C01815=1076.234,414.000,-108.664,176.398,32.358,155.824
C01816=1076.246,414.386,-108.731,176.405,32.374,155.827
C01817=1076.257,414.773,-108.798,176.414,32.390,155.831
C01818=1076.269,415.159,-108.866,176.422,32.405,155.834
C01819=1076.276,415.405,-108.908,176.427,32.415,155.836
C01820=1076.283,415.651,-108.952,176.432,32.425,155.839
C01821=1076.291,415.898,-108.995,176.438,32.436,155.841
C01822=1076.298,416.143,-109.038,176.442,32.446,155.843
C01823=1076.305,416.389,-109.080,176.447,32.456,155.846
C01824=1076.313,416.636,-109.124,176.453,32.466,155.848
C01825=1076.320,416.882,-109.167,176.458,32.477,155.850
C01826=1076.327,417.128,-109.210,176.463,32.487,155.853
C01827=1076.334,417.374,-109.253,176.469,32.497,155.855
C01828=1076.342,417.620,-109.297,176.474,32.507,155.857
C01829=1076.349,417.867,-109.340,176.480,32.518,155.859
C01830=1076.356,418.112,-109.383,176.485,32.529,155.862
C01831=1076.363,418.358,-109.426,176.489,32.539,155.864
C01832=1076.371,418.605,-109.470,176.495,32.549,155.867
C01833=1076.378,418.850,-109.513,176.500,32.560,155.869
C01834=1076.386,419.097,-109.557,176.506,32.571,155.871
C01835=1076.392,419.343,-109.600,176.511,32.581,155.874
C01836=1076.400,419.589,-109.644,176.517,32.592,155.876
C01837=1076.408,419.835,-109.688,176.522,32.602,155.879
C01838=1076.415,420.081,-109.731,176.528,32.613,155.881
C01839=1076.423,420.327,-109.775,176.533,32.624,155.883
C01840=1076.430,420.573,-109.818,176.539,32.635,155.886
C01841=1076.438,420.819,-109.861,176.544,32.645,155.888
C01842=1076.446,421.066,-109.905,176.550,32.656,155.891
C01843=1076.453,421.311,-109.949,176.555,32.667,155.893
C01844=1076.460,421.557,-109.993,176.561,32.677,155.896
C01845=1076.468,421.804,-110.037,176.566,32.688,155.898
C01846=1076.475,422.049,-110.080,176.572,32.700,155.901
C01847=1076.482,422.295,-110.125,176.577,32.710,155.903
C01848=1076.490,422.542,-110.169,176.583,32.721,155.906
C01849=1076.498,422.787,-110.213,176.589,32.733,155.908
C01850=1076.505,423.034,-110.257,176.594,32.744,155.911
C01851=1076.513,423.279,-110.301,176.600,32.755,155.913
C01852=1076.520,423.525,-110.344,176.605,32.766,155.916
C01853=1076.527,423.771,-110.389,176.611,32.777,155.918
C01854=1076.535,424.017,-110.433,176.617,32.789,155.921
C01855=1076.542,424.263,-110.478,176.622,32.800,155.924
C01856=1076.550,424.508,-110.522,176.628,32.811,155.926
C01857=1076.557,424.755,-110.566,176.634,32.823,155.929
C01858=1076.565,425.001,-110.610,176.639,32.834,155.931
C01859=1076.573,425.247,-110.655,176.645,32.845,155.934
C01860=1076.580,425.493,-110.700,176.651,32.857,155.937
C01861=1076.588,425.738,-110.744,176.656,32.868,155.939
C01862=1076.595,425.984,-110.788,176.662,32.879,155.942
C01863=1076.604,426.253,-110.836,176.668,32.892,155.945
C01864=1076.612,426.521,-110.885,176.675,32.905,155.948
C01865=1076.620,426.788,-110.934,176.681,32.917,155.951
C01866=1076.629,427.057,-110.983,176.687,32.930,155.953
C01867=1076.636,427.303,-111.027,176.693,32.942,155.956
C01868=1076.644,427.548,-111.072,176.699,32.954,155.959
C01869=1076.652,427.794,-111.117,176.705,32.965,155.962
C01870=1076.660,428.040,-111.161,176.711,32.977,155.964
C01871=1076.667,428.286,-111.206,176.717,32.989,155.967
C01872=1076.674,428.532,-111.251,176.723,33.001,155.970
C01873=1076.682,428.778,-111.297,176.729,33.013,155.973
C01874=1076.690,429.023,-111.341,176.735,33.024,155.975
C01875=1076.697,429.270,-111.386,176.740,33.037,155.978
C01876=1076.705,429.515,-111.432,176.746,33.048,155.981
C01877=1076.713,429.761,-111.476,176.753,33.061,155.984
C01878=1076.721,430.006,-111.522,176.759,33.073,155.987
C01879=1076.728,430.252,-111.566,176.765,33.085,155.989
C01880=1076.736,430.498,-111.612,176.771,33.097,155.992
C01881=1076.744,430.744,-111.657,176.777,33.109,155.995
C01882=1076.752,430.989,-111.702,176.783,33.122,155.998
C01883=1076.760,431.235,-111.748,176.790,33.134,156.001
C01884=1076.767,431.481,-111.793,176.796,33.146,156.004
C01885=1076.775,431.726,-111.838,176.802,33.159,156.007
C01886=1076.784,431.972,-111.884,176.808,33.171,156.010
C01887=1076.791,432.218,-111.929,176.814,33.184,156.013
C01888=1076.799,432.464,-111.975,176.820,33.196,156.015
C01889=1076.806,432.709,-112.020,176.826,33.209,156.018
C01890=1076.814,432.955,-112.066,176.832,33.221,156.021
C01891=1076.822,433.201,-112.112,176.839,33.234,156.024
C01892=1076.830,433.446,-112.158,176.846,33.247,156.027
C01893=1076.837,433.692,-112.203,176.852,33.259,156.030
C01894=1076.845,433.937,-112.249,176.858,33.272,156.033
C01895=1076.853,434.183,-112.295,176.865,33.285,156.036
C01896=1076.861,434.429,-112.341,176.871,33.298,156.040
C01897=1076.869,434.673,-112.387,176.877,33.311,156.043
C01898=1076.877,434.920,-112.433,176.883,33.323,156.046
C01899=1076.885,435.165,-112.479,176.890,33.337,156.049
C01900=1076.892,435.410,-112.524,176.896,33.349,156.052
C01901=1076.901,435.656,-112.571,176.902,33.363,156.055
C01902=1076.909,435.901,-112.617,176.910,33.376,156.058
C01903=1076.917,436.147,-112.663,176.916,33.389,156.061
C01904=1076.925,436.392,-112.709,176.922,33.402,156.064
C01905=1076.932,436.639,-112.756,176.929,33.415,156.067
C01906=1076.940,436.884,-112.802,176.935,33.429,156.071
C01907=1076.948,437.130,-112.848,176.943,33.442,156.074
C01908=1076.956,437.374,-112.894,176.949,33.455,156.077
C01909=1076.965,437.620,-112.941,176.955,33.468,156.080
C01910=1076.973,437.865,-112.987,176.962,33.482,156.083
C01911=1076.981,438.111,-113.033,176.969,33.495,156.086
C01912=1076.989,438.356,-113.080,176.976,33.509,156.090
C01913=1076.998,438.601,-113.127,176.982,33.523,156.093
C01914=1077.005,438.848,-113.173,176.988,33.536,156.096
C01915=1077.013,439.093,-113.220,176.996,33.550,156.099
C01916=1077.022,439.338,-113.266,177.002,33.563,156.103
C01917=1077.030,439.584,-113.313,177.009,33.577,156.106
C01918=1077.037,439.829,-113.360,177.016,33.591,156.109
C01919=1077.048,440.127,-113.418,177.024,33.608,156.113
C01920=1077.057,440.426,-113.474,177.033,33.625,156.118
C01921=1077.067,440.725,-113.531,177.041,33.642,156.122
C01922=1077.078,441.024,-113.589,177.050,33.659,156.126
C01923=1077.086,441.269,-113.635,177.056,33.673,156.129
C01924=1077.093,441.515,-113.683,177.064,33.688,156.133
C01925=1077.102,441.760,-113.730,177.070,33.702,156.136
C01926=1077.110,442.006,-113.777,177.078,33.716,156.140
C01927=1077.119,442.250,-113.825,177.085,33.730,156.143
C01928=1077.127,442.496,-113.872,177.092,33.745,156.147
C01929=1077.135,442.740,-113.919,177.099,33.759,156.150
C01930=1077.143,442.986,-113.967,177.106,33.773,156.154
C01931=1077.152,443.231,-114.014,177.113,33.788,156.157
C01932=1077.159,443.477,-114.061,177.121,33.803,156.161
C01933=1077.168,443.722,-114.109,177.127,33.817,156.164
C01934=1077.176,443.967,-114.157,177.135,33.832,156.168
C01935=1077.185,444.213,-114.204,177.143,33.847,156.171
C01936=1077.193,444.458,-114.252,177.149,33.861,156.175
C01937=1077.201,444.703,-114.300,177.157,33.876,156.179
C01938=1077.210,444.948,-114.347,177.164,33.891,156.182
C01939=1077.218,445.193,-114.395,177.171,33.906,156.186
C01940=1077.226,445.438,-114.443,177.179,33.921,156.190
C01941=1077.235,445.683,-114.491,177.186,33.936,156.193
C01942=1077.243,445.928,-114.539,177.194,33.951,156.197
C01943=1077.251,446.174,-114.587,177.202,33.966,156.201
C01944=1077.259,446.419,-114.635,177.209,33.981,156.204
C01945=1077.269,446.664,-114.683,177.216,33.996,156.208
C01946=1077.277,446.909,-114.731,177.223,34.012,156.212
C01947=1077.285,447.154,-114.779,177.230,34.027,156.216
C01948=1077.293,447.399,-114.827,177.237,34.042,156.219
C01949=1077.303,447.644,-114.876,177.242,34.057,156.223
C01950=1077.311,447.890,-114.924,177.248,34.072,156.227
C01951=1077.320,448.134,-114.973,177.254,34.087,156.231
C01952=1077.329,448.379,-115.020,177.260,34.103,156.235
C01953=1077.337,448.624,-115.069,177.265,34.117,156.238
C01954=1077.345,448.869,-115.117,177.270,34.133,156.242
C01955=1077.355,449.113,-115.164,177.275,34.147,156.246
C01956=1077.367,449.358,-115.211,177.280,34.161,156.249
C01957=1077.380,449.603,-115.257,177.284,34.174,156.253
C01958=1077.394,449.849,-115.303,177.288,34.187,156.256
C01959=1077.034,449.844,-115.535,177.267,34.346,156.298
C01960=1077.019,449.599,-115.489,177.263,34.333,156.295
C01961=1077.006,449.354,-115.444,177.258,34.320,156.291
C01962=1076.995,449.108,-115.397,177.253,34.306,156.288
C01963=1076.985,448.864,-115.349,177.248,34.292,156.284
C01964=1076.976,448.619,-115.302,177.243,34.277,156.280
C01965=1076.967,448.374,-115.252,177.237,34.261,156.277
C01966=1076.959,448.130,-115.204,177.232,34.246,156.273
C01967=1076.949,447.885,-115.156,177.226,34.231,156.269
C01968=1076.941,447.640,-115.107,177.220,34.216,156.265
C01969=1076.933,447.395,-115.059,177.213,34.201,156.261
C01970=1076.924,447.150,-115.010,177.206,34.185,156.258
C01971=1076.916,446.904,-114.962,177.199,34.170,156.254
C01972=1076.907,446.660,-114.915,177.192,34.156,156.250
C01973=1076.899,446.415,-114.866,177.185,34.140,156.246
C01974=1076.891,446.170,-114.818,177.177,34.125,156.243
C01975=1076.881,445.924,-114.770,177.170,34.110,156.239
C01976=1076.873,445.679,-114.722,177.162,34.095,156.235
C01977=1076.865,445.434,-114.674,177.155,34.080,156.231
C01978=1076.857,445.189,-114.625,177.147,34.065,156.228
C01979=1076.848,444.944,-114.578,177.139,34.050,156.224
C01980=1076.840,444.699,-114.530,177.132,34.035,156.220
C01981=1076.832,444.453,-114.483,177.125,34.020,156.217
C01982=1076.823,444.208,-114.435,177.117,34.005,156.213
C01983=1076.815,443.963,-114.387,177.110,33.991,156.210
C01984=1076.806,443.718,-114.340,177.102,33.976,156.206
C01985=1076.798,443.473,-114.292,177.096,33.962,156.202
C01986=1076.789,443.228,-114.245,177.088,33.947,156.199
C01987=1076.781,442.982,-114.197,177.081,33.932,156.195
C01988=1076.773,442.737,-114.149,177.073,33.918,156.192
C01989=1076.765,442.492,-114.102,177.067,33.904,156.188
C01990=1076.756,442.246,-114.054,177.059,33.889,156.185
C01991=1076.748,442.001,-114.007,177.052,33.875,156.181
C01992=1076.740,441.756,-113.959,177.045,33.861,156.178
C01993=1076.732,441.511,-113.913,177.038,33.847,156.174
C01994=1076.723,441.265,-113.866,177.030,33.833,156.171
C01995=1076.715,441.020,-113.818,177.024,33.818,156.168
C01996=1076.706,440.739,-113.764,177.015,33.802,156.164
C01997=1076.696,440.456,-113.711,177.007,33.786,156.160
C01998=1076.687,440.175,-113.656,177.000,33.770,156.156
C01999=1076.678,439.894,-113.603,176.991,33.754,156.152
C02000=1076.669,439.649,-113.556,176.984,33.740,156.149
C02001=1076.661,439.403,-113.509,176.978,33.727,156.145
C02002=1076.653,439.158,-113.462,176.970,33.713,156.142
C02003=1076.645,438.912,-113.416,176.964,33.699,156.139
C02004=1076.636,438.667,-113.369,176.957,33.686,156.136
C02005=1076.628,438.421,-113.322,176.950,33.672,156.132
C02006=1076.620,438.176,-113.275,176.943,33.658,156.129
C02007=1076.612,437.930,-113.229,176.937,33.645,156.126
C02008=1076.604,437.685,-113.183,176.930,33.631,156.123
C02009=1076.596,437.440,-113.136,176.923,33.618,156.119
C02010=1076.587,437.194,-113.089,176.916,33.605,156.116
C02011=1076.580,436.949,-113.044,176.910,33.591,156.113
C02012=1076.571,436.703,-112.997,176.903,33.578,156.110
C02013=1076.564,436.458,-112.951,176.896,33.565,156.107
C02014=1076.556,436.212,-112.904,176.889,33.552,156.103
C02015=1076.548,435.967,-112.858,176.883,33.538,156.100
C02016=1076.539,435.721,-112.812,176.877,33.526,156.097
C02017=1076.532,435.476,-112.766,176.870,33.513,156.094
C02018=1076.523,435.230,-112.719,176.864,33.499,156.091
C02019=1076.516,434.985,-112.674,176.857,33.487,156.088
C02020=1076.508,434.739,-112.628,176.850,33.473,156.085
C02021=1076.499,434.494,-112.581,176.844,33.461,156.082
C02022=1076.492,434.248,-112.536,176.837,33.448,156.079
C02023=1076.484,434.003,-112.490,176.831,33.435,156.076
C02024=1076.476,433.757,-112.444,176.824,33.422,156.073
C02025=1076.468,433.511,-112.398,176.818,33.410,156.070
C02026=1076.461,433.266,-112.353,176.812,33.397,156.067
C02027=1076.452,433.020,-112.307,176.805,33.384,156.064
C02028=1076.445,432.774,-112.261,176.799,33.371,156.061
C02029=1076.437,432.529,-112.215,176.793,33.359,156.058
C02030=1076.429,432.283,-112.170,176.786,33.346,156.055
C02031=1076.421,432.037,-112.124,176.780,33.334,156.052
C02032=1076.414,431.792,-112.078,176.774,33.321,156.049
C02033=1076.406,431.546,-112.032,176.768,33.309,156.046
C02034=1076.398,431.301,-111.988,176.761,33.297,156.043
C02035=1076.390,431.055,-111.942,176.755,33.285,156.040
C02036=1076.382,430.809,-111.896,176.749,33.272,156.037
C02037=1076.375,430.563,-111.851,176.742,33.260,156.034
C02038=1076.366,430.318,-111.806,176.736,33.248,156.032
C02039=1076.359,430.073,-111.761,176.731,33.236,156.029
C02040=1076.351,429.826,-111.716,176.725,33.223,156.026
C02041=1076.344,429.581,-111.670,176.719,33.211,156.023
C02042=1076.336,429.335,-111.626,176.712,33.199,156.020
C02043=1076.328,429.090,-111.580,176.706,33.187,156.017
C02044=1076.320,428.843,-111.535,176.700,33.176,156.015
C02045=1076.312,428.597,-111.491,176.694,33.163,156.012
C02046=1076.304,428.352,-111.445,176.688,33.151,156.009
C02047=1076.297,428.106,-111.400,176.682,33.140,156.006
C02048=1076.290,427.860,-111.355,176.676,33.128,156.004
C02049=1076.282,427.614,-111.311,176.670,33.116,156.001
C02050=1076.274,427.368,-111.266,176.664,33.104,155.998
C02051=1076.266,427.122,-111.221,176.659,33.092,155.995
C02052=1076.258,426.853,-111.172,176.651,33.080,155.993
C02053=1076.249,426.583,-111.123,176.645,33.067,155.990
C02054=1076.240,426.314,-111.074,176.639,33.054,155.987
C02055=1076.232,426.044,-111.025,176.632,33.042,155.984
C02056=1076.225,425.798,-110.980,176.627,33.031,155.981
C02057=1076.217,425.552,-110.936,176.621,33.019,155.978
C02058=1076.210,425.307,-110.891,176.615,33.007,155.976
C02059=1076.202,425.061,-110.847,176.609,32.996,155.973
C02060=1076.194,424.814,-110.803,176.603,32.985,155.970
C02061=1076.187,424.568,-110.759,176.597,32.973,155.968
C02062=1076.179,424.323,-110.714,176.592,32.962,155.965
C02063=1076.171,424.077,-110.669,176.586,32.951,155.963
C02064=1076.164,423.831,-110.626,176.580,32.939,155.960
C02065=1076.157,423.585,-110.581,176.575,32.929,155.958
C02066=1076.149,423.339,-110.537,176.569,32.917,155.955
C02067=1076.141,423.093,-110.493,176.564,32.906,155.952
C02068=1076.134,422.847,-110.449,176.558,32.895,155.950
C02069=1076.127,422.601,-110.405,176.552,32.884,155.947
C02070=1076.119,422.355,-110.361,176.547,32.873,155.945
C02071=1076.112,422.109,-110.317,176.540,32.862,155.942
C02072=1076.104,421.863,-110.273,176.535,32.851,155.940
C02073=1076.096,421.617,-110.229,176.529,32.840,155.937
C02074=1076.090,421.371,-110.185,176.524,32.829,155.935
C02075=1076.082,421.125,-110.141,176.518,32.818,155.932
C02076=1076.074,420.879,-110.097,176.513,32.807,155.930
C02077=1076.067,420.634,-110.054,176.507,32.797,155.927
C02078=1076.059,420.387,-110.010,176.502,32.786,155.925
C02079=1076.051,420.141,-109.967,176.496,32.775,155.923
C02080=1076.044,419.895,-109.923,176.491,32.764,155.920
C02081=1076.037,419.648,-109.879,176.485,32.754,155.918
C02082=1076.030,419.403,-109.836,176.480,32.743,155.915
C02083=1076.022,419.156,-109.792,176.474,32.733,155.913
C02084=1076.014,418.910,-109.749,176.469,32.722,155.911
C02085=1076.007,418.664,-109.705,176.463,32.711,155.908
C02086=1076.000,418.418,-109.662,176.458,32.701,155.906
C02087=1075.992,418.172,-109.618,176.453,32.691,155.903
C02088=1075.985,417.926,-109.575,176.447,32.680,155.901
C02089=1075.977,417.680,-109.532,176.442,32.670,155.899
C02090=1075.970,417.434,-109.488,176.436,32.660,155.896
C02091=1075.963,417.188,-109.445,176.431,32.649,155.894
C02092=1075.956,416.942,-109.402,176.426,32.639,155.892
C02093=1075.948,416.696,-109.359,176.421,32.628,155.889
C02094=1075.941,416.450,-109.315,176.416,32.618,155.887
C02095=1075.933,416.203,-109.272,176.411,32.608,155.885
C02096=1075.926,415.957,-109.229,176.405,32.598,155.882
C02097=1075.919,415.712,-109.186,176.400,32.587,155.880
C02098=1075.911,415.465,-109.143,176.395,32.578,155.878
C02099=1075.904,415.219,-109.100,176.389,32.567,155.876
C02100=1075.897,414.973,-109.057,176.384,32.557,155.873
C02101=1075.890,414.726,-109.014,176.379,32.547,155.871
C02102=1075.882,414.480,-108.972,176.374,32.537,155.869
C02103=1075.875,414.234,-108.929,176.368,32.527,155.867
C02104=1075.867,413.988,-108.885,176.363,32.517,155.864
C02105=1075.861,413.741,-108.843,176.358,32.507,155.862
C02106=1075.853,413.495,-108.801,176.354,32.497,155.860
C02107=1075.845,413.249,-108.757,176.348,32.487,155.858
C02108=1075.838,412.997,-108.714,176.343,32.478,155.856
C02109=1075.831,412.745,-108.671,176.338,32.468,155.853
C02110=1075.823,412.493,-108.627,176.332,32.458,155.851
C02111=1075.816,412.241,-108.583,176.327,32.448,155.849
C02112=1075.809,411.995,-108.541,176.322,32.438,155.847
C02113=1075.801,411.749,-108.499,176.317,32.429,155.845
C02114=1075.794,411.502,-108.456,176.312,32.419,155.842
C02115=1075.787,411.255,-108.413,176.307,32.409,155.840
C02116=1075.779,411.010,-108.371,176.302,32.399,155.838
C02117=1075.773,410.763,-108.329,176.297,32.390,155.836
C02118=1075.766,410.517,-108.286,176.292,32.380,155.834
C02119=1075.758,410.271,-108.244,176.287,32.371,155.832
C02120=1075.751,410.025,-108.202,176.282,32.361,155.830
C02121=1075.744,409.778,-108.159,176.277,32.352,155.828
C02122=1075.736,409.532,-108.117,176.272,32.342,155.826
C02123=1075.730,409.285,-108.075,176.267,32.333,155.823
C02124=1075.722,409.039,-108.033,176.262,32.323,155.821
C02125=1075.715,408.793,-107.991,176.257,32.314,155.819
C02126=1075.708,408.546,-107.948,176.252,32.305,155.817
C02127=1075.701,408.300,-107.907,176.247,32.295,155.815
C02128=1075.694,408.053,-107.864,176.243,32.286,155.813
C02129=1075.687,407.807,-107.822,176.238,32.276,155.811
C02130=1075.680,407.561,-107.781,176.233,32.268,155.809
C02131=1075.673,407.314,-107.738,176.228,32.258,155.807
C02132=1075.667,407.068,-107.697,176.223,32.249,155.805
C02133=1075.660,406.822,-107.655,176.219,32.240,155.803
C02134=1075.652,406.575,-107.613,176.214,32.230,155.801
C02135=1075.645,406.329,-107.571,176.209,32.221,155.799
C02136=1075.638,406.083,-107.530,176.204,32.213,155.797
C02137=1075.631,405.837,-107.488,176.199,32.203,155.795
C02138=1075.624,405.590,-107.446,176.195,32.194,155.793
C02139=1075.617,405.343,-107.405,176.190,32.185,155.791
C02140=1075.609,405.097,-107.363,176.185,32.176,155.789
C02141=1075.603,404.850,-107.321,176.180,32.167,155.787
C02142=1075.595,404.604,-107.280,176.175,32.158,155.785
C02143=1075.589,404.358,-107.239,176.171,32.149,155.783
C02144=1075.582,404.111,-107.196,176.166,32.141,155.781
C02145=1075.575,403.865,-107.155,176.162,32.132,155.779
C02146=1075.567,403.618,-107.114,176.157,32.123,155.777
C02147=1075.560,403.372,-107.073,176.152,32.114,155.775
C02148=1075.554,403.125,-107.031,176.148,32.105,155.774
C02149=1075.547,402.879,-106.990,176.143,32.096,155.772
C02150=1075.539,402.632,-106.949,176.138,32.088,155.770
C02151=1075.532,402.386,-106.907,176.133,32.079,155.768
C02152=1075.525,402.139,-106.866,176.129,32.070,155.766
C02153=1075.518,401.893,-106.825,176.124,32.062,155.764
C02154=1075.512,401.646,-106.784,176.120,32.053,155.762
C02155=1075.504,401.400,-106.742,176.115,32.044,155.760
C02156=1075.498,401.154,-106.701,176.111,32.035,155.759
C02157=1075.490,400.907,-106.660,176.106,32.027,155.757
C02158=1075.483,400.661,-106.619,176.101,32.019,155.755
C02159=1075.477,400.414,-106.579,176.096,32.010,155.753
C02160=1075.470,400.179,-106.539,176.093,32.002,155.751
C02161=1075.464,399.943,-106.500,176.088,31.994,155.750
C02162=1075.456,399.708,-106.461,176.084,31.986,155.748
C02163=1075.450,399.472,-106.422,176.079,31.978,155.746
C02164=1075.443,399.237,-106.382,176.075,31.970,155.744
C02165=1075.437,399.001,-106.343,176.071,31.961,155.743
C02166=1075.430,398.765,-106.305,176.066,31.953,155.741
C02167=1075.421,398.432,-106.250,176.060,31.942,155.738
C02168=1075.414,398.186,-106.209,176.056,31.934,155.737
C02169=1075.407,397.939,-106.168,176.051,31.925,155.735
C02170=1075.400,397.692,-106.127,176.047,31.917,155.733
C02171=1075.393,397.446,-106.087,176.043,31.909,155.731
C02172=1075.386,397.199,-106.046,176.038,31.901,155.730
C02173=1075.380,396.953,-106.006,176.033,31.892,155.728
C02174=1075.372,396.706,-105.964,176.029,31.885,155.726
C02175=1075.366,396.460,-105.924,176.025,31.876,155.724
C02176=1075.358,396.213,-105.884,176.020,31.868,155.723
C02177=1075.351,395.967,-105.843,176.015,31.860,155.721
C02178=1075.345,395.720,-105.803,176.012,31.852,155.719
C02179=1075.338,395.473,-105.763,176.007,31.844,155.717
C02180=1075.331,395.227,-105.722,176.002,31.835,155.716
C02181=1075.324,394.980,-105.681,175.998,31.827,155.714
C02182=1075.317,394.734,-105.642,175.994,31.819,155.712
C02183=1075.311,394.487,-105.602,175.989,31.811,155.711
C02184=1075.304,394.240,-105.561,175.985,31.803,155.709
C02185=1075.297,393.994,-105.520,175.981,31.795,155.707
C02186=1075.290,393.747,-105.480,175.976,31.787,155.705
C02187=1075.283,393.501,-105.440,175.972,31.779,155.704
C02188=1075.277,393.254,-105.400,175.968,31.772,155.702
C02189=1075.269,393.007,-105.360,175.963,31.764,155.701
C02190=1075.263,392.761,-105.320,175.959,31.756,155.699
C02191=1075.256,392.514,-105.280,175.954,31.748,155.697
C02192=1075.249,392.268,-105.240,175.950,31.740,155.695
C02193=1075.242,392.021,-105.200,175.946,31.732,155.694
C02194=1075.236,391.774,-105.160,175.941,31.724,155.692
C02195=1075.229,391.528,-105.120,175.937,31.716,155.691
C02196=1075.222,391.282,-105.080,175.933,31.709,155.689
C02197=1075.215,391.034,-105.041,175.928,31.701,155.687
C02198=1075.208,390.788,-105.001,175.924,31.694,155.686
C02199=1075.201,390.541,-104.961,175.920,31.686,155.684
C02200=1075.195,390.295,-104.921,175.915,31.678,155.683
C02201=1075.187,390.048,-104.881,175.912,31.670,155.681
C02202=1075.181,389.801,-104.842,175.907,31.663,155.679
C02203=1075.174,389.555,-104.802,175.902,31.655,155.678
C02204=1075.167,389.308,-104.763,175.899,31.648,155.676
C02205=1075.161,389.061,-104.723,175.894,31.640,155.675
C02206=1075.153,388.814,-104.683,175.890,31.633,155.673
C02207=1075.147,388.568,-104.643,175.886,31.625,155.671
C02208=1075.140,388.321,-104.604,175.881,31.617,155.670
C02209=1075.133,388.075,-104.565,175.877,31.610,155.668
C02210=1075.127,387.828,-104.525,175.873,31.603,155.667
C02211=1075.120,387.582,-104.486,175.869,31.595,155.665
C02212=1075.113,387.335,-104.447,175.864,31.588,155.664
C02213=1075.106,387.088,-104.407,175.861,31.580,155.662
C02214=1075.100,386.841,-104.368,175.856,31.573,155.661
C02215=1075.093,386.595,-104.328,175.852,31.565,155.659
C02216=1075.086,386.354,-104.290,175.848,31.558,155.658
C02217=1075.080,386.114,-104.252,175.844,31.551,155.656
C02218=1075.074,385.874,-104.214,175.839,31.544,155.655
C02219=1075.067,385.633,-104.175,175.836,31.537,155.653
C02220=1075.060,385.394,-104.137,175.832,31.530,155.652
C02221=1075.054,385.153,-104.099,175.828,31.522,155.650
C02222=1075.047,384.913,-104.060,175.824,31.515,155.649
C02223=1075.041,384.672,-104.022,175.819,31.508,155.647
C02224=1075.034,384.425,-103.983,175.816,31.501,155.646
C02225=1075.027,384.179,-103.944,175.811,31.494,155.644
C02226=1075.021,383.932,-103.905,175.807,31.486,155.643
C02227=1075.015,383.686,-103.866,175.804,31.479,155.641
C02228=1075.008,383.439,-103.827,175.799,31.472,155.640
C02229=1075.001,383.192,-103.788,175.795,31.464,155.638
C02230=1074.995,382.945,-103.749,175.791,31.457,155.637
C02231=1074.988,382.698,-103.710,175.787,31.451,155.635
C02232=1074.981,382.451,-103.671,175.782,31.443,155.634
C02233=1074.974,382.204,-103.632,175.779,31.436,155.632
C02234=1074.968,381.957,-103.593,175.774,31.429,155.631
C02235=1074.962,381.711,-103.555,175.771,31.422,155.629
C02236=1074.955,381.464,-103.516,175.766,31.415,155.628
C02237=1074.949,381.218,-103.477,175.762,31.408,155.627
C02238=1074.942,380.971,-103.438,175.759,31.401,155.625
C02239=1074.935,380.724,-103.399,175.754,31.394,155.624
C02240=1074.928,380.477,-103.360,175.750,31.387,155.622
C02241=1074.922,380.230,-103.322,175.746,31.380,155.621
C02242=1074.915,379.983,-103.283,175.742,31.373,155.619
C02243=1074.909,379.737,-103.245,175.739,31.366,155.618
C02244=1074.902,379.490,-103.206,175.734,31.359,155.617
C02245=1074.895,379.243,-103.169,175.730,31.352,155.615
C02246=1074.888,378.996,-103.130,175.726,31.345,155.614
C02247=1074.881,378.749,-103.091,175.722,31.338,155.612
C02248=1074.875,378.502,-103.053,175.719,31.332,155.611
C02249=1074.868,378.256,-103.014,175.714,31.324,155.610
C02250=1074.862,378.008,-102.976,175.710,31.318,155.608
C02251=1074.855,377.761,-102.937,175.706,31.311,155.607
C02252=1074.849,377.515,-102.899,175.702,31.304,155.605
C02253=1074.842,377.268,-102.861,175.698,31.298,155.604
C02254=1074.835,377.021,-102.822,175.694,31.291,155.603
C02255=1074.829,376.773,-102.784,175.690,31.284,155.601
C02256=1074.823,376.527,-102.745,175.687,31.277,155.600
C02257=1074.815,376.280,-102.708,175.682,31.270,155.599
C02258=1074.809,376.033,-102.670,175.678,31.264,155.597
C02259=1074.803,375.787,-102.631,175.675,31.257,155.596
C02260=1074.796,375.539,-102.593,175.670,31.250,155.595
C02261=1074.789,375.292,-102.554,175.667,31.243,155.593
C02262=1074.783,375.046,-102.516,175.663,31.237,155.592
C02263=1074.777,374.798,-102.478,175.658,31.230,155.590
C02264=1074.771,374.551,-102.441,175.655,31.223,155.589
C02265=1074.764,374.305,-102.402,175.651,31.217,155.588
C02266=1074.757,374.057,-102.364,175.648,31.210,155.586
C02267=1074.751,373.811,-102.326,175.643,31.203,155.585
C02268=1074.745,373.563,-102.288,175.639,31.197,155.584
C02269=1074.738,373.317,-102.250,175.636,31.191,155.583
C02270=1074.731,373.070,-102.212,175.631,31.183,155.581
C02271=1074.725,372.823,-102.174,175.628,31.177,155.580
C02272=1074.718,372.597,-102.140,175.624,31.171,155.579
C02273=1074.713,372.371,-102.105,175.620,31.165,155.578
C02274=1074.707,372.145,-102.072,175.617,31.159,155.576
C02275=1074.701,371.920,-102.037,175.613,31.153,155.575
C02276=1074.695,371.694,-102.002,175.610,31.148,155.574
C02277=1074.689,371.468,-101.968,175.607,31.142,155.573
C02278=1074.683,371.243,-101.933,175.603,31.136,155.572
C02279=1074.677,371.017,-101.898,175.600,31.130,155.570
C02280=1074.670,370.770,-101.861,175.596,31.124,155.569
C02281=1074.664,370.523,-101.823,175.591,31.117,155.568
C02282=1074.657,370.276,-101.787,175.588,31.111,155.567
C02283=1074.651,370.028,-101.748,175.584,31.104,155.565
C02284=1074.644,369.782,-101.711,175.581,31.098,155.564
C02285=1074.638,369.535,-101.673,175.576,31.092,155.563
C02286=1074.631,369.288,-101.636,175.572,31.086,155.562
C02287=1074.625,369.041,-101.598,175.569,31.079,155.560
C02288=1074.618,368.794,-101.561,175.565,31.073,155.559
C02289=1074.612,368.546,-101.523,175.562,31.067,155.558
C02290=1074.605,368.300,-101.486,175.557,31.060,155.557
C02291=1074.600,368.052,-101.449,175.554,31.054,155.555
C02292=1074.592,367.805,-101.412,175.550,31.048,155.554
C02293=1074.586,367.559,-101.374,175.546,31.041,155.553
C02294=1074.579,367.311,-101.337,175.543,31.035,155.552
C02295=1074.574,367.064,-101.299,175.538,31.029,155.550
C02296=1074.567,366.818,-101.262,175.535,31.023,155.549
C02297=1074.561,366.570,-101.225,175.531,31.016,155.548
C02298=1074.554,366.323,-101.188,175.527,31.010,155.547
C02299=1074.548,366.076,-101.151,175.524,31.004,155.546
C02300=1074.541,365.829,-101.113,175.519,30.998,155.544
C02301=1074.536,365.581,-101.076,175.516,30.992,155.543
C02302=1074.529,365.335,-101.039,175.512,30.985,155.542
C02303=1074.522,365.087,-101.002,175.509,30.979,155.541
C02304=1074.516,364.840,-100.964,175.505,30.973,155.540
C02305=1074.510,364.593,-100.928,175.501,30.967,155.538
C02306=1074.503,364.345,-100.891,175.498,30.961,155.537
C02307=1074.497,364.099,-100.853,175.493,30.955,155.536
C02308=1074.491,363.852,-100.817,175.490,30.949,155.535
C02309=1074.484,363.604,-100.780,175.486,30.943,155.534
C02310=1074.477,363.357,-100.743,175.483,30.937,155.532
C02311=1074.471,363.110,-100.706,175.479,30.931,155.531
C02312=1074.465,362.862,-100.669,175.475,30.925,155.530
C02313=1074.458,362.615,-100.632,175.472,30.919,155.529
C02314=1074.452,362.368,-100.596,175.467,30.913,155.528
C02315=1074.445,362.122,-100.559,175.464,30.907,155.527
C02316=1074.438,361.874,-100.522,175.460,30.901,155.525
C02317=1074.433,361.627,-100.485,175.457,30.895,155.524
C02318=1074.426,361.380,-100.449,175.453,30.889,155.523
C02319=1074.420,361.133,-100.412,175.449,30.883,155.522
C02320=1074.413,360.885,-100.375,175.446,30.877,155.521
C02321=1074.407,360.638,-100.339,175.442,30.871,155.520
C02322=1074.400,360.391,-100.302,175.439,30.865,155.518
C02323=1074.394,360.144,-100.266,175.434,30.859,155.517
C02324=1074.388,359.896,-100.229,175.431,30.853,155.516
C02325=1074.382,359.649,-100.193,175.427,30.848,155.515
C02326=1074.375,359.401,-100.156,175.424,30.842,155.514
C02327=1074.369,359.154,-100.119,175.420,30.836,155.513
C02328=1074.363,358.937,-100.088,175.417,30.831,155.512
C02329=1074.357,358.720,-100.055,175.414,30.826,155.511
C02330=1074.352,358.503,-100.024,175.410,30.821,155.510
C02331=1074.346,358.285,-99.991,175.407,30.815,155.509
C02332=1074.340,358.068,-99.960,175.404,30.810,155.508
C02333=1074.335,357.850,-99.928,175.401,30.805,155.507
C02334=1074.329,357.633,-99.895,175.398,30.800,155.506
C02335=1074.324,357.416,-99.863,175.395,30.795,155.505
C02336=1074.317,357.168,-99.827,175.391,30.790,155.504
C02337=1074.311,356.921,-99.791,175.387,30.783,155.503
C02338=1074.305,356.674,-99.754,175.383,30.778,155.502
C02339=1074.298,356.426,-99.718,175.380,30.772,155.501
C02340=1074.292,356.179,-99.682,175.376,30.766,155.499
C02341=1074.285,355.932,-99.646,175.373,30.760,155.498
C02342=1074.279,355.685,-99.610,175.369,30.755,155.497
C02343=1074.273,355.437,-99.574,175.366,30.750,155.496
C02344=1074.267,355.190,-99.538,175.362,30.744,155.495
C02345=1074.260,354.943,-99.501,175.358,30.738,155.494
C02346=1074.254,354.696,-99.466,175.355,30.732,155.493
C02347=1074.248,354.448,-99.429,175.351,30.727,155.492
C02348=1074.242,354.201,-99.393,175.348,30.721,155.491
C02349=1074.236,353.954,-99.357,175.344,30.715,155.490
C02350=1074.229,353.706,-99.322,175.341,30.710,155.489
C02351=1074.222,353.459,-99.285,175.337,30.704,155.488
C02352=1074.216,353.212,-99.250,175.334,30.698,155.486
C02353=1074.210,352.965,-99.213,175.330,30.693,155.485
C02354=1074.204,352.717,-99.177,175.326,30.687,155.484
C02355=1074.198,352.469,-99.142,175.323,30.682,155.483
C02356=1074.191,352.223,-99.106,175.319,30.676,155.482
C02357=1074.185,351.975,-99.070,175.316,30.670,155.481
C02358=1074.179,351.727,-99.034,175.312,30.665,155.480
C02359=1074.172,351.480,-98.999,175.309,30.659,155.479
C02360=1074.166,351.233,-98.963,175.305,30.654,155.478
C02361=1074.160,350.985,-98.927,175.302,30.648,155.477
C02362=1074.153,350.738,-98.892,175.298,30.643,155.476
C02363=1074.147,350.491,-98.856,175.295,30.638,155.475
C02364=1074.141,350.243,-98.820,175.292,30.632,155.474
C02365=1074.134,349.996,-98.785,175.288,30.627,155.473
C02366=1074.128,349.749,-98.749,175.285,30.621,155.472
C02367=1074.122,349.501,-98.714,175.281,30.616,155.471
C02368=1074.116,349.254,-98.678,175.278,30.610,155.470
C02369=1074.109,349.007,-98.642,175.274,30.605,155.469
C02370=1074.102,348.759,-98.607,175.271,30.600,155.468
C02371=1074.096,348.511,-98.571,175.267,30.594,155.467
C02372=1074.091,348.265,-98.536,175.264,30.589,155.466
C02373=1074.084,348.017,-98.501,175.260,30.583,155.465
C02374=1074.078,347.769,-98.465,175.256,30.578,155.464
C02375=1074.071,347.522,-98.430,175.253,30.572,155.463
C02376=1074.065,347.274,-98.394,175.249,30.567,155.462
C02377=1074.059,347.027,-98.359,175.247,30.562,155.461
C02378=1074.053,346.780,-98.324,175.243,30.556,155.460
C02379=1074.046,346.533,-98.288,175.240,30.551,155.459
C02380=1074.041,346.284,-98.253,175.236,30.545,155.458
C02381=1074.035,346.037,-98.218,175.233,30.540,155.457
C02382=1074.029,345.790,-98.183,175.229,30.535,155.456
C02383=1074.022,345.543,-98.148,175.226,30.529,155.455
C02384=1074.017,345.327,-98.117,175.223,30.525,155.454
C02385=1074.011,345.112,-98.086,175.219,30.520,155.453
C02386=1074.005,344.896,-98.056,175.217,30.516,155.452
C02387=1074.001,344.680,-98.025,175.214,30.511,155.451
C02388=1073.995,344.464,-97.994,175.211,30.506,155.450
C02389=1073.989,344.249,-97.963,175.208,30.502,155.449
C02390=1073.984,344.033,-97.933,175.205,30.497,155.449
C02391=1073.979,343.817,-97.902,175.202,30.492,155.448
C02392=1073.972,343.570,-97.867,175.198,30.487,155.447
C02393=1073.966,343.321,-97.832,175.195,30.482,155.446
C02394=1073.960,343.075,-97.797,175.192,30.477,155.445
C02395=1073.953,342.827,-97.762,175.189,30.472,155.444
C02396=1073.947,342.579,-97.728,175.185,30.467,155.443
C02397=1073.941,342.332,-97.693,175.181,30.462,155.442
C02398=1073.935,342.084,-97.658,175.178,30.456,155.441
C02399=1073.928,341.837,-97.623,175.174,30.451,155.440
C02400=1073.922,341.590,-97.589,175.171,30.446,155.439
C02401=1073.916,341.342,-97.553,175.168,30.441,155.438
C02402=1073.910,341.094,-97.519,175.165,30.436,155.437
C02403=1073.904,340.848,-97.484,175.161,30.430,155.436
C02404=1073.897,340.600,-97.450,175.158,30.425,155.435
C02405=1073.891,340.352,-97.414,175.154,30.420,155.434
C02406=1073.885,340.105,-97.380,175.152,30.415,155.433
C02407=1073.879,339.857,-97.345,175.148,30.410,155.432
C02408=1073.873,339.610,-97.311,175.145,30.405,155.432
C02409=1073.867,339.362,-97.276,175.141,30.399,155.431
C02410=1073.860,339.114,-97.240,175.137,30.394,155.430
C02411=1073.854,338.867,-97.206,175.134,30.389,155.429
C02412=1073.848,338.620,-97.171,175.131,30.384,155.428
C02413=1073.842,338.372,-97.137,175.128,30.379,155.427
C02414=1073.836,338.124,-97.102,175.124,30.374,155.426
C02415=1073.830,337.877,-97.068,175.121,30.369,155.425
C02416=1073.823,337.629,-97.033,175.118,30.364,155.424
C02417=1073.817,337.382,-96.999,175.115,30.359,155.423
C02418=1073.811,337.134,-96.965,175.111,30.354,155.422
C02419=1073.805,336.886,-96.930,175.108,30.349,155.421
C02420=1073.799,336.639,-96.896,175.104,30.344,155.420
C02421=1073.792,336.391,-96.862,175.102,30.339,155.419
C02422=1073.786,336.144,-96.827,175.098,30.334,155.418
C02423=1073.780,335.896,-96.792,175.095,30.329,155.418
C02424=1073.774,335.649,-96.758,175.091,30.324,155.417
C02425=1073.767,335.401,-96.724,175.088,30.319,155.416
C02426=1073.761,335.154,-96.690,175.085,30.314,155.415
C02427=1073.755,334.906,-96.656,175.081,30.309,155.414
C02428=1073.749,334.658,-96.621,175.078,30.304,155.413
C02429=1073.743,334.410,-96.587,175.075,30.299,155.412
C02430=1073.737,334.163,-96.553,175.072,30.294,155.411
C02431=1073.731,333.916,-96.519,175.068,30.289,155.410
C02432=1073.724,333.668,-96.485,175.065,30.284,155.409
C02433=1073.719,333.421,-96.450,175.062,30.279,155.409
C02434=1073.712,333.173,-96.416,175.059,30.274,155.408
C02435=1073.706,332.925,-96.382,175.055,30.269,155.407
C02436=1073.700,332.677,-96.348,175.052,30.264,155.406
C02437=1073.693,332.430,-96.315,175.049,30.260,155.405
C02438=1073.688,332.182,-96.281,175.046,30.255,155.404
C02439=1073.681,331.934,-96.246,175.042,30.250,155.403
C02440=1073.676,331.716,-96.217,175.039,30.245,155.402
C02441=1073.671,331.498,-96.186,175.037,30.241,155.402
C02442=1073.666,331.280,-96.156,175.034,30.237,155.401
C02443=1073.660,331.062,-96.126,175.031,30.232,155.400
C02444=1073.655,330.844,-96.096,175.028,30.228,155.399
C02445=1073.649,330.625,-96.067,175.025,30.224,155.399
C02446=1073.643,330.407,-96.037,175.022,30.219,155.398
C02447=1073.638,330.189,-96.008,175.019,30.216,155.397
C02448=1073.631,329.940,-95.974,175.016,30.211,155.396
C02449=1073.625,329.693,-95.940,175.013,30.206,155.395
C02450=1073.618,329.445,-95.906,175.010,30.201,155.395
C02451=1073.613,329.198,-95.873,175.006,30.196,155.394
C02452=1073.606,328.951,-95.839,175.004,30.192,155.393
C02453=1073.600,328.703,-95.805,175.000,30.187,155.392
C02454=1073.593,328.455,-95.772,174.997,30.182,155.391
C02455=1073.588,328.208,-95.738,174.994,30.178,155.390
C02456=1073.581,327.959,-95.705,174.990,30.172,155.389
C02457=1073.575,327.712,-95.671,174.987,30.168,155.389
C02458=1073.569,327.464,-95.637,174.984,30.163,155.388
C02459=1073.562,327.217,-95.604,174.981,30.159,155.387
C02460=1073.557,326.969,-95.570,174.977,30.154,155.386
C02461=1073.550,326.722,-95.537,174.975,30.149,155.385
C02462=1073.544,326.474,-95.503,174.971,30.144,155.384
C02463=1073.538,326.225,-95.470,174.968,30.140,155.384
C02464=1073.532,325.978,-95.436,174.965,30.135,155.383
C02465=1073.525,325.731,-95.404,174.962,30.130,155.382
C02466=1073.519,325.483,-95.369,174.958,30.126,155.381
C02467=1073.513,325.235,-95.336,174.956,30.121,155.380
C02468=1073.507,324.987,-95.303,174.952,30.116,155.379
C02469=1073.500,324.740,-95.270,174.950,30.111,155.378
C02470=1073.495,324.492,-95.236,174.946,30.107,155.378
C02471=1073.488,324.244,-95.203,174.943,30.102,155.377
C02472=1073.482,323.996,-95.170,174.940,30.098,155.376
C02473=1073.476,323.749,-95.136,174.936,30.093,155.375
C02474=1073.470,323.501,-95.103,174.933,30.088,155.374
C02475=1073.464,323.254,-95.070,174.930,30.084,155.374
C02476=1073.458,323.006,-95.037,174.927,30.079,155.373
C02477=1073.451,322.758,-95.003,174.924,30.074,155.372
C02478=1073.446,322.510,-94.970,174.921,30.070,155.371
C02479=1073.439,322.262,-94.937,174.917,30.065,155.370
C02480=1073.434,322.015,-94.904,174.915,30.060,155.369
C02481=1073.428,321.767,-94.871,174.911,30.055,155.368
C02482=1073.421,321.519,-94.838,174.909,30.051,155.368
C02483=1073.416,321.271,-94.805,174.905,30.046,155.367
C02484=1073.409,321.024,-94.772,174.902,30.041,155.366
C02485=1073.404,320.777,-94.738,174.899,30.037,155.365
C02486=1073.397,320.529,-94.705,174.896,30.032,155.364
C02487=1073.392,320.281,-94.672,174.893,30.027,155.364
C02488=1073.385,320.033,-94.639,174.890,30.023,155.363
C02489=1073.379,319.785,-94.606,174.887,30.019,155.362
C02490=1073.373,319.537,-94.573,174.884,30.013,155.361
C02491=1073.367,319.290,-94.540,174.880,30.009,155.360
C02492=1073.361,319.042,-94.507,174.877,30.005,155.360
C02493=1073.355,318.794,-94.475,174.874,30.000,155.359
C02494=1073.349,318.546,-94.442,174.871,29.995,155.358
C02495=1073.343,318.298,-94.409,174.868,29.991,155.357
C02496=1073.338,318.077,-94.380,174.865,29.986,155.356
C02497=1073.333,317.856,-94.349,174.863,29.982,155.356
C02498=1073.328,317.634,-94.321,174.860,29.978,155.355
C02499=1073.322,317.413,-94.291,174.858,29.974,155.354
C02500=1073.317,317.192,-94.262,174.854,29.970,155.354
C02501=1073.311,316.970,-94.233,174.852,29.966,155.353
C02502=1073.306,316.749,-94.203,174.849,29.962,155.352
C02503=1073.300,316.527,-94.174,174.846,29.958,155.351
C02504=1073.295,316.280,-94.141,174.843,29.953,155.350
C02505=1073.289,316.031,-94.109,174.840,29.949,155.350
C02506=1073.283,315.784,-94.076,174.837,29.944,155.349
C02507=1073.278,315.537,-94.043,174.834,29.939,155.348
C02508=1073.272,315.288,-94.011,174.831,29.935,155.347
C02509=1073.265,315.041,-93.978,174.828,29.930,155.346
C02510=1073.260,314.793,-93.945,174.825,29.926,155.346
C02511=1073.254,314.545,-93.912,174.822,29.921,155.345
C02512=1073.248,314.297,-93.880,174.819,29.916,155.344
C02513=1073.241,314.049,-93.847,174.816,29.912,155.343
C02514=1073.235,313.801,-93.815,174.813,29.908,155.343
C02515=1073.229,313.554,-93.782,174.810,29.904,155.342
C02516=1073.223,313.305,-93.750,174.807,29.899,155.341
C02517=1073.216,313.058,-93.718,174.804,29.895,155.340
C02518=1073.210,312.810,-93.686,174.801,29.890,155.339
C02519=1073.204,312.563,-93.654,174.798,29.886,155.339
C02520=1073.198,312.315,-93.622,174.795,29.881,155.338
C02521=1073.192,312.067,-93.589,174.792,29.877,155.337
C02522=1073.186,311.819,-93.557,174.788,29.873,155.336
C02523=1073.180,311.571,-93.524,174.786,29.868,155.336
C02524=1073.173,311.323,-93.493,174.782,29.864,155.335
C02525=1073.167,311.076,-93.460,174.780,29.860,155.334
C02526=1073.161,310.828,-93.428,174.776,29.855,155.333
C02527=1073.155,310.579,-93.396,174.774,29.851,155.333
C02528=1073.149,310.333,-93.364,174.770,29.847,155.332
C02529=1073.143,310.084,-93.332,174.768,29.842,155.331
C02530=1073.136,309.836,-93.300,174.764,29.838,155.330
C02531=1073.130,309.589,-93.268,174.762,29.833,155.330
C02532=1073.124,309.341,-93.236,174.758,29.829,155.329
C02533=1073.119,309.093,-93.204,174.756,29.825,155.328
C02534=1073.112,308.846,-93.171,174.752,29.820,155.327
C02535=1073.106,308.598,-93.140,174.750,29.816,155.327
C02536=1073.100,308.349,-93.108,174.746,29.811,155.326
C02537=1073.094,308.101,-93.076,174.744,29.807,155.325
C02538=1073.088,307.854,-93.043,174.740,29.803,155.324
C02539=1073.082,307.606,-93.011,174.738,29.798,155.324
C02540=1073.075,307.358,-92.980,174.735,29.794,155.323
C02541=1073.070,307.111,-92.948,174.732,29.790,155.322
C02542=1073.064,306.862,-92.916,174.729,29.786,155.321
C02543=1073.058,306.614,-92.884,174.726,29.781,155.321
C02544=1073.051,306.367,-92.852,174.723,29.777,155.320
C02545=1073.045,306.119,-92.820,174.720,29.772,155.319
C02546=1073.040,305.871,-92.788,174.717,29.768,155.318
C02547=1073.034,305.623,-92.756,174.714,29.764,155.318
C02548=1073.027,305.376,-92.725,174.711,29.759,155.317
C02549=1073.021,305.128,-92.693,174.709,29.755,155.316
C02550=1073.015,304.879,-92.661,174.705,29.751,155.315
C02551=1073.009,304.632,-92.630,174.702,29.746,155.315
C02552=1073.004,304.412,-92.601,174.700,29.743,155.314
C02553=1072.999,304.193,-92.573,174.697,29.739,155.313
C02554=1072.993,303.973,-92.545,174.695,29.735,155.313
C02555=1072.988,303.753,-92.518,174.692,29.731,155.312
C02556=1072.983,303.533,-92.489,174.689,29.727,155.311
C02557=1072.978,303.314,-92.461,174.686,29.723,155.311
C02558=1072.973,303.094,-92.433,174.684,29.719,155.310
C02559=1072.967,302.874,-92.405,174.681,29.715,155.309
C02560=1072.961,302.626,-92.373,174.678,29.711,155.309
C02561=1072.955,302.378,-92.342,174.676,29.707,155.308
C02562=1072.949,302.130,-92.310,174.672,29.703,155.307
C02563=1072.944,301.882,-92.279,174.670,29.698,155.306
C02564=1072.937,301.635,-92.247,174.666,29.694,155.306
C02565=1072.932,301.387,-92.216,174.664,29.690,155.305
C02566=1072.926,301.139,-92.184,174.661,29.685,155.304
C02567=1072.920,300.891,-92.153,174.658,29.681,155.303
C02568=1072.914,300.643,-92.121,174.655,29.677,155.303
C02569=1072.909,300.395,-92.090,174.652,29.672,155.302
C02570=1072.902,300.147,-92.058,174.649,29.668,155.301
C02571=1072.897,299.899,-92.027,174.647,29.664,155.301
C02572=1072.890,299.651,-91.996,174.643,29.659,155.300
C02573=1072.885,299.404,-91.964,174.641,29.655,155.299
C02574=1072.879,299.155,-91.933,174.638,29.651,155.298
C02575=1072.873,298.908,-91.902,174.635,29.647,155.298
C02576=1072.867,298.660,-91.870,174.632,29.642,155.297
C02577=1072.862,298.411,-91.839,174.630,29.638,155.296
C02578=1072.856,298.164,-91.808,174.626,29.634,155.295
C02579=1072.850,297.916,-91.776,174.624,29.629,155.295
C02580=1072.844,297.668,-91.745,174.621,29.625,155.294
C02581=1072.838,297.420,-91.713,174.618,29.621,155.293
C02582=1072.832,297.172,-91.683,174.615,29.616,155.292
C02583=1072.826,296.924,-91.651,174.612,29.612,155.292
C02584=1072.820,296.676,-91.621,174.609,29.608,155.291
C02585=1072.814,296.428,-91.589,174.607,29.604,155.290
C02586=1072.809,296.180,-91.558,174.603,29.599,155.290
C02587=1072.802,295.932,-91.527,174.601,29.596,155.289
C02588=1072.796,295.684,-91.496,174.598,29.591,155.288
C02589=1072.791,295.437,-91.465,174.595,29.587,155.287
C02590=1072.784,295.188,-91.434,174.592,29.583,155.287
C02591=1072.779,294.941,-91.404,174.590,29.579,155.286
C02592=1072.773,294.692,-91.372,174.586,29.575,155.285
C02593=1072.767,294.445,-91.341,174.584,29.570,155.285
C02594=1072.760,294.197,-91.310,174.581,29.566,155.284
C02595=1072.754,293.949,-91.279,174.578,29.562,155.283
C02596=1072.748,293.701,-91.249,174.575,29.558,155.283
C02597=1072.743,293.452,-91.218,174.573,29.553,155.282
C02598=1072.737,293.205,-91.187,174.569,29.549,155.281
C02599=1072.730,292.956,-91.156,174.567,29.546,155.280
C02600=1072.724,292.709,-91.126,174.564,29.541,155.280
C02601=1072.719,292.461,-91.094,174.562,29.537,155.279
C02602=1072.713,292.213,-91.063,174.558,29.533,155.278
C02603=1072.707,291.965,-91.033,174.556,29.529,155.278
C02604=1072.701,291.717,-91.003,174.553,29.525,155.277
C02605=1072.694,291.468,-90.972,174.550,29.520,155.276
C02606=1072.689,291.221,-90.940,174.547,29.516,155.276
C02607=1072.683,290.973,-90.910,174.545,29.512,155.275
C02608=1072.678,290.761,-90.884,174.542,29.509,155.274
C02609=1072.672,290.548,-90.858,174.540,29.505,155.274
C02610=1072.667,290.336,-90.832,174.537,29.501,155.273
C02611=1072.662,290.123,-90.805,174.534,29.498,155.273
C02612=1072.657,289.911,-90.779,174.533,29.494,155.272
C02613=1072.652,289.698,-90.753,174.530,29.491,155.271
C02614=1072.647,289.486,-90.727,174.528,29.487,155.271
C02615=1072.642,289.274,-90.700,174.525,29.484,155.270
C02616=1072.637,289.026,-90.670,174.523,29.479,155.269
C02617=1072.630,288.777,-90.639,174.520,29.475,155.269
C02618=1072.624,288.529,-90.609,174.517,29.471,155.268
C02619=1072.618,288.282,-90.579,174.514,29.467,155.267
C02620=1072.612,288.033,-90.548,174.512,29.463,155.267
C02621=1072.606,287.785,-90.518,174.509,29.459,155.266
C02622=1072.600,287.537,-90.487,174.506,29.455,155.265
C02623=1072.594,287.289,-90.456,174.503,29.451,155.265
C02624=1072.588,287.041,-90.426,174.501,29.447,155.264
C02625=1072.583,286.793,-90.396,174.497,29.443,155.263
C02626=1072.576,286.545,-90.367,174.495,29.439,155.263
C02627=1072.570,286.297,-90.336,174.492,29.435,155.262
C02628=1072.564,286.049,-90.306,174.490,29.430,155.261
C02629=1072.558,285.801,-90.275,174.486,29.426,155.261
C02630=1072.552,285.553,-90.245,174.484,29.422,155.260
C02631=1072.546,285.304,-90.215,174.481,29.418,155.259
C02632=1072.540,285.056,-90.185,174.479,29.414,155.258
C02633=1072.535,284.808,-90.154,174.475,29.410,155.258
C02634=1072.529,284.560,-90.124,174.473,29.406,155.257
C02635=1072.523,284.313,-90.094,174.470,29.402,155.256
C02636=1072.517,284.063,-90.064,174.468,29.398,155.256
C02637=1072.510,283.816,-90.034,174.465,29.394,155.255
C02638=1072.504,283.568,-90.003,174.462,29.390,155.254
C02639=1072.499,283.320,-89.974,174.459,29.386,155.254
C02640=1072.493,283.072,-89.943,174.457,29.381,155.253
C02641=1072.487,282.824,-89.913,174.454,29.377,155.252
C02642=1072.482,282.576,-89.883,174.451,29.373,155.252
C02643=1072.475,282.327,-89.853,174.448,29.369,155.251
C02644=1072.469,282.080,-89.823,174.446,29.365,155.250
C02645=1072.463,281.831,-89.793,174.443,29.361,155.250
C02646=1072.457,281.583,-89.763,174.441,29.357,155.249
C02647=1072.452,281.335,-89.733,174.437,29.353,155.248
C02648=1072.446,281.087,-89.703,174.435,29.349,155.248
C02649=1072.441,280.839,-89.673,174.432,29.345,155.247
C02650=1072.434,280.591,-89.644,174.430,29.341,155.246
C02651=1072.429,280.343,-89.614,174.427,29.337,155.246
C02652=1072.422,280.094,-89.583,174.424,29.332,155.245
C02653=1072.417,279.846,-89.554,174.421,29.328,155.244
C02654=1072.410,279.598,-89.524,174.419,29.324,155.244
C02655=1072.405,279.350,-89.494,174.416,29.321,155.243
C02656=1072.398,279.102,-89.464,174.414,29.317,155.242
C02657=1072.392,278.854,-89.435,174.410,29.312,155.242
C02658=1072.387,278.606,-89.405,174.408,29.309,155.241
C02659=1072.380,278.358,-89.375,174.405,29.304,155.240
C02660=1072.375,278.109,-89.346,174.403,29.300,155.239
C02661=1072.369,277.862,-89.315,174.400,29.296,155.239
C02662=1072.363,277.613,-89.286,174.398,29.292,155.238
C02663=1072.357,277.365,-89.257,174.395,29.288,155.238
C02664=1072.347,276.950,-89.207,174.390,29.282,155.236
C02665=1072.337,276.536,-89.157,174.386,29.275,155.235
C02666=1072.327,276.121,-89.108,174.381,29.268,155.234
C02667=1072.317,275.706,-89.059,174.377,29.261,155.233
C02668=1072.312,275.458,-89.029,174.374,29.257,155.232
C02669=1072.305,275.210,-89.000,174.372,29.254,155.232
C02670=1072.300,274.962,-88.970,174.369,29.249,155.231
C02671=1072.294,274.714,-88.941,174.367,29.245,155.230
C02672=1072.288,274.465,-88.911,174.364,29.241,155.230
C02673=1072.282,274.217,-88.882,174.361,29.237,155.229
C02674=1072.276,273.969,-88.853,174.359,29.233,155.228
C02675=1072.270,273.721,-88.823,174.356,29.229,155.228
C02676=1072.264,273.473,-88.793,174.354,29.225,155.227
C02677=1072.258,273.225,-88.764,174.351,29.221,155.226
C02678=1072.253,272.976,-88.734,174.349,29.218,155.226
C02679=1072.246,272.728,-88.705,174.345,29.213,155.225
C02680=1072.241,272.480,-88.676,174.343,29.209,155.224
C02681=1072.235,272.232,-88.647,174.340,29.205,155.224
C02682=1072.228,271.983,-88.618,174.338,29.201,155.223
C02683=1072.223,271.735,-88.588,174.335,29.197,155.222
C02684=1072.217,271.487,-88.559,174.333,29.193,155.222
C02685=1072.210,271.239,-88.530,174.330,29.189,155.221
C02686=1072.205,270.990,-88.500,174.327,29.185,155.221
C02687=1072.199,270.743,-88.472,174.324,29.181,155.220
C02688=1072.194,270.494,-88.442,174.322,29.177,155.219
C02689=1072.187,270.246,-88.413,174.319,29.173,155.219
C02690=1072.181,269.998,-88.385,174.317,29.169,155.218
C02691=1072.176,269.749,-88.355,174.314,29.166,155.217
C02692=1072.170,269.501,-88.326,174.312,29.162,155.217
C02693=1072.163,269.253,-88.297,174.309,29.158,155.216
C02694=1072.157,269.005,-88.268,174.307,29.154,155.215
C02695=1072.152,268.756,-88.238,174.303,29.150,155.215
C02696=1072.146,268.509,-88.210,174.301,29.146,155.214
C02697=1072.140,268.260,-88.181,174.298,29.142,155.213
C02698=1072.134,268.012,-88.152,174.296,29.138,155.213
C02699=1072.128,267.763,-88.123,174.294,29.134,155.212
C02700=1072.122,267.515,-88.094,174.291,29.129,155.211
C02701=1072.116,267.267,-88.065,174.289,29.125,155.211
C02702=1072.110,267.018,-88.036,174.286,29.121,155.210
C02703=1072.104,266.771,-88.008,174.284,29.118,155.209
C02704=1072.099,266.522,-87.979,174.281,29.114,155.209
C02705=1072.093,266.274,-87.950,174.279,29.110,155.208
C02706=1072.087,266.026,-87.921,174.275,29.106,155.207
C02707=1072.081,265.777,-87.892,174.273,29.102,155.207
C02708=1072.075,265.530,-87.864,174.270,29.098,155.206
C02709=1072.069,265.281,-87.834,174.268,29.094,155.206
C02710=1072.063,265.032,-87.806,174.265,29.090,155.205
C02711=1072.057,264.784,-87.777,174.263,29.086,155.204
C02712=1072.051,264.536,-87.748,174.260,29.082,155.204
C02713=1072.046,264.288,-87.720,174.258,29.078,155.203
C02714=1072.039,264.040,-87.691,174.255,29.074,155.202
C02715=1072.034,263.791,-87.662,174.253,29.070,155.202
C02716=1072.024,263.380,-87.615,174.249,29.064,155.201
C02717=1072.014,262.969,-87.567,174.245,29.057,155.200
C02718=1072.004,262.558,-87.520,174.241,29.051,155.198
C02719=1071.994,262.146,-87.473,174.235,29.044,155.197
C02720=1071.988,261.898,-87.444,174.233,29.040,155.197
C02721=1071.982,261.649,-87.416,174.231,29.036,155.196
C02722=1071.976,261.400,-87.387,174.228,29.033,155.196
C02723=1071.969,261.152,-87.359,174.226,29.029,155.195
C02724=1071.964,260.904,-87.331,174.223,29.025,155.194
C02725=1071.957,260.656,-87.302,174.221,29.021,155.194
C02726=1071.951,260.407,-87.274,174.218,29.017,155.193
C02727=1071.946,260.159,-87.245,174.216,29.013,155.192
C02728=1071.940,259.911,-87.217,174.213,29.009,155.192
C02729=1071.933,259.663,-87.189,174.211,29.005,155.191
C02730=1071.927,259.414,-87.160,174.208,29.002,155.191
C02731=1071.922,259.166,-87.133,174.206,28.998,155.190
C02732=1071.916,258.918,-87.103,174.203,28.994,155.189
C02733=1071.910,258.669,-87.075,174.201,28.990,155.189
C02734=1071.904,258.420,-87.047,174.198,28.986,155.188
C02735=1071.898,258.173,-87.019,174.196,28.982,155.187
C02736=1071.891,257.924,-86.990,174.193,28.978,155.187
C02737=1071.886,257.676,-86.962,174.191,28.974,155.186
C02738=1071.880,257.428,-86.934,174.189,28.970,155.185
C02739=1071.874,257.179,-86.906,174.186,28.966,155.185
C02740=1071.868,256.930,-86.878,174.184,28.962,155.184
C02741=1071.862,256.682,-86.850,174.181,28.958,155.183
C02742=1071.856,256.434,-86.821,174.179,28.955,155.183
C02743=1071.851,256.186,-86.793,174.176,28.951,155.182
C02744=1071.844,255.938,-86.765,174.174,28.947,155.182
C02745=1071.838,255.689,-86.737,174.171,28.943,155.181
C02746=1071.833,255.441,-86.709,174.169,28.939,155.180
C02747=1071.827,255.192,-86.681,174.166,28.935,155.180
C02748=1071.821,254.944,-86.653,174.164,28.931,155.179
C02749=1071.815,254.696,-86.625,174.161,28.927,155.178
C02750=1071.809,254.447,-86.597,174.159,28.923,155.178
C02751=1071.803,254.199,-86.569,174.157,28.919,155.177
C02752=1071.797,253.950,-86.541,174.154,28.915,155.176
C02753=1071.791,253.702,-86.513,174.152,28.911,155.176
C02754=1071.785,253.454,-86.485,174.149,28.907,155.175
C02755=1071.780,253.206,-86.457,174.147,28.903,155.175
C02756=1071.773,252.957,-86.429,174.144,28.899,155.174
C02757=1071.768,252.709,-86.401,174.142,28.895,155.173
C02758=1071.762,252.460,-86.373,174.139,28.891,155.173
C02759=1071.756,252.212,-86.345,174.137,28.888,155.172
C02760=1071.750,251.964,-86.317,174.134,28.884,155.171
C02761=1071.744,251.715,-86.290,174.132,28.880,155.171
C02762=1071.739,251.466,-86.262,174.130,28.876,155.170
C02763=1071.733,251.219,-86.234,174.127,28.872,155.169
C02764=1071.727,250.970,-86.206,174.125,28.868,155.169
C02765=1071.722,250.722,-86.178,174.122,28.864,155.168
C02766=1071.716,250.473,-86.150,174.120,28.860,155.167
C02767=1071.710,250.225,-86.123,174.117,28.856,155.167
C02768=1071.700,249.811,-86.076,174.113,28.849,155.166
C02769=1071.690,249.397,-86.030,174.109,28.843,155.165
C02770=1071.681,248.983,-85.984,174.105,28.836,155.164
C02771=1071.672,248.570,-85.937,174.102,28.830,155.162
C02772=1071.666,248.321,-85.910,174.100,28.826,155.162
C02773=1071.660,248.073,-85.882,174.097,28.822,155.161
C02774=1071.654,247.824,-85.854,174.095,28.818,155.161
C02775=1071.649,247.575,-85.827,174.092,28.814,155.160
C02776=1071.643,247.327,-85.799,174.090,28.810,155.159
C02777=1071.637,247.079,-85.772,174.087,28.806,155.159
C02778=1071.631,246.830,-85.744,174.085,28.802,155.158
C02779=1071.625,246.582,-85.717,174.083,28.798,155.157
C02780=1071.619,246.334,-85.689,174.080,28.794,155.157
C02781=1071.614,246.085,-85.662,174.078,28.790,155.156
C02782=1071.608,245.837,-85.634,174.075,28.786,155.155
C02783=1071.602,245.588,-85.607,174.073,28.782,155.155
C02784=1071.596,245.340,-85.579,174.070,28.778,155.154
C02785=1071.590,245.091,-85.552,174.069,28.774,155.153
C02786=1071.585,244.843,-85.524,174.066,28.770,155.153
C02787=1071.579,244.594,-85.497,174.064,28.766,155.152
C02788=1071.572,244.346,-85.470,174.062,28.762,155.151
C02789=1071.567,244.098,-85.442,174.059,28.758,155.151
C02790=1071.561,243.849,-85.415,174.057,28.755,155.150
C02791=1071.556,243.601,-85.387,174.054,28.751,155.150
C02792=1071.550,243.352,-85.361,174.052,28.747,155.149
C02793=1071.543,243.104,-85.333,174.049,28.743,155.148
C02794=1071.538,242.855,-85.306,174.047,28.739,155.148
C02795=1071.532,242.607,-85.278,174.045,28.735,155.147
C02796=1071.526,242.358,-85.251,174.043,28.731,155.146
C02797=1071.521,242.110,-85.224,174.041,28.727,155.146
C02798=1071.515,241.862,-85.197,174.038,28.723,155.145
C02799=1071.508,241.613,-85.170,174.036,28.719,155.145
C02800=1071.503,241.364,-85.143,174.033,28.715,155.144
C02801=1071.497,241.116,-85.115,174.031,28.711,155.143
C02802=1071.491,240.867,-85.088,174.029,28.707,155.143
C02803=1071.485,240.619,-85.062,174.026,28.704,155.142
C02804=1071.479,240.371,-85.035,174.024,28.700,155.141
C02805=1071.473,240.122,-85.007,174.022,28.696,155.141
C02806=1071.468,239.873,-84.980,174.020,28.692,155.140
C02807=1071.462,239.625,-84.953,174.017,28.688,155.139
C02808=1071.455,239.376,-84.926,174.015,28.684,155.139
C02809=1071.449,239.128,-84.899,174.012,28.680,155.138
C02810=1071.444,238.880,-84.872,174.010,28.676,155.138
C02811=1071.438,238.632,-84.846,174.008,28.672,155.137
C02812=1071.431,238.383,-84.819,174.005,28.668,155.136
C02813=1071.426,238.134,-84.791,174.004,28.665,155.136
C02814=1071.421,237.886,-84.765,174.001,28.661,155.135
C02815=1071.415,237.637,-84.738,173.999,28.657,155.134
C02816=1071.408,237.389,-84.710,173.996,28.653,155.134
C02817=1071.402,237.140,-84.684,173.994,28.649,155.133
C02818=1071.397,236.892,-84.657,173.992,28.645,155.133
C02819=1071.391,236.644,-84.630,173.989,28.641,155.132
C02820=1071.381,236.222,-84.585,173.986,28.634,155.131
C02821=1071.371,235.802,-84.540,173.982,28.628,155.130
C02822=1071.361,235.382,-84.494,173.978,28.621,155.129
C02823=1071.352,234.961,-84.449,173.974,28.614,155.128
C02824=1071.346,234.713,-84.423,173.972,28.610,155.127
C02825=1071.340,234.464,-84.396,173.969,28.606,155.126
C02826=1071.334,234.216,-84.369,173.968,28.603,155.126
C02827=1071.328,233.967,-84.342,173.965,28.599,155.125
C02828=1071.322,233.719,-84.316,173.963,28.595,155.124
C02829=1071.317,233.471,-84.289,173.961,28.591,155.124
C02830=1071.311,233.222,-84.262,173.958,28.587,155.123
C02831=1071.304,232.973,-84.235,173.956,28.583,155.122
C02832=1071.299,232.725,-84.209,173.954,28.579,155.122
C02833=1071.293,232.476,-84.182,173.952,28.575,155.121
C02834=1071.287,232.228,-84.156,173.949,28.571,155.120
C02835=1071.282,231.979,-84.130,173.947,28.567,155.120
C02836=1071.276,231.731,-84.103,173.945,28.563,155.119
C02837=1071.270,231.482,-84.076,173.942,28.559,155.119
C02838=1071.264,231.234,-84.050,173.941,28.555,155.118
C02839=1071.258,230.984,-84.023,173.938,28.551,155.117
C02840=1071.252,230.736,-83.997,173.936,28.547,155.117
C02841=1071.246,230.488,-83.971,173.934,28.543,155.116
C02842=1071.240,230.240,-83.944,173.931,28.540,155.115
C02843=1071.235,229.991,-83.918,173.930,28.536,155.115
C02844=1071.229,229.742,-83.891,173.927,28.532,155.114
C02845=1071.223,229.494,-83.865,173.925,28.528,155.114
C02846=1071.218,229.245,-83.839,173.922,28.524,155.113
C02847=1071.211,228.997,-83.813,173.920,28.520,155.112
C02848=1071.205,228.748,-83.786,173.919,28.516,155.112
C02849=1071.199,228.499,-83.760,173.916,28.512,155.111
C02850=1071.194,228.250,-83.733,173.914,28.508,155.110
C02851=1071.187,228.002,-83.707,173.911,28.504,155.110
C02852=1071.182,227.753,-83.681,173.909,28.500,155.109
C02853=1071.176,227.505,-83.655,173.908,28.497,155.108
C02854=1071.170,227.256,-83.629,173.905,28.493,155.108
C02855=1071.164,227.008,-83.603,173.903,28.489,155.107
C02856=1071.158,226.760,-83.576,173.900,28.485,155.107
C02857=1071.153,226.511,-83.550,173.898,28.481,155.106
C02858=1071.146,226.263,-83.524,173.897,28.477,155.105
C02859=1071.141,226.014,-83.498,173.894,28.473,155.105
C02860=1071.135,225.765,-83.471,173.892,28.469,155.104
C02861=1071.129,225.517,-83.446,173.889,28.465,155.103
C02862=1071.123,225.268,-83.419,173.888,28.461,155.103
C02863=1071.117,225.019,-83.393,173.886,28.457,155.102
C02864=1071.111,224.771,-83.367,173.883,28.453,155.101
C02865=1071.105,224.522,-83.341,173.881,28.449,155.101
C02866=1071.100,224.273,-83.315,173.878,28.445,155.100
C02867=1071.093,224.025,-83.289,173.877,28.441,155.099
C02868=1071.088,223.776,-83.264,173.875,28.437,155.099
C02869=1071.082,223.528,-83.237,173.872,28.433,155.098
C02870=1071.076,223.279,-83.212,173.870,28.429,155.098
C02871=1071.071,223.030,-83.186,173.868,28.425,155.097
C02872=1071.065,222.816,-83.163,173.866,28.422,155.096
C02873=1071.061,222.602,-83.140,173.864,28.419,155.096
C02874=1071.056,222.388,-83.118,173.863,28.416,155.095
C02875=1071.050,222.173,-83.096,173.860,28.412,155.095
C02876=1071.045,221.960,-83.074,173.859,28.408,155.094
C02877=1071.041,221.745,-83.051,173.857,28.405,155.094
C02878=1071.035,221.531,-83.029,173.855,28.402,155.093
C02879=1071.030,221.316,-83.006,173.854,28.398,155.092
C02880=1071.024,221.067,-82.981,173.851,28.394,155.092
C02881=1071.018,220.818,-82.955,173.849,28.390,155.091
C02882=1071.013,220.571,-82.929,173.846,28.386,155.091
C02883=1071.007,220.322,-82.903,173.845,28.382,155.090
C02884=1071.001,220.073,-82.878,173.843,28.378,155.089
C02885=1070.995,219.824,-82.852,173.840,28.374,155.089
C02886=1070.989,219.576,-82.826,173.838,28.370,155.088
C02887=1070.983,219.328,-82.801,173.836,28.367,155.087
C02888=1070.977,219.079,-82.775,173.834,28.363,155.087
C02889=1070.971,218.830,-82.750,173.832,28.359,155.086
C02890=1070.966,218.581,-82.724,173.830,28.355,155.086
C02891=1070.959,218.332,-82.698,173.828,28.351,155.085
C02892=1070.953,218.084,-82.673,173.825,28.347,155.084
C02893=1070.948,217.836,-82.647,173.823,28.343,155.084
C02894=1070.942,217.587,-82.621,173.822,28.339,155.083
C02895=1070.936,217.338,-82.595,173.819,28.335,155.082
C02896=1070.930,217.090,-82.570,173.817,28.331,155.082
C02897=1070.924,216.841,-82.545,173.814,28.327,155.081
C02898=1070.918,216.592,-82.519,173.813,28.324,155.080
C02899=1070.912,216.343,-82.493,173.811,28.319,155.080
C02900=1070.907,216.095,-82.468,173.808,28.315,155.079
C02901=1070.901,215.847,-82.443,173.807,28.312,155.078
C02902=1070.895,215.598,-82.417,173.805,28.308,155.078
C02903=1070.889,215.349,-82.391,173.802,28.304,155.077
C02904=1070.883,215.100,-82.366,173.801,28.300,155.077
C02905=1070.878,214.852,-82.341,173.798,28.296,155.076
C02906=1070.872,214.603,-82.315,173.796,28.291,155.075
C02907=1070.866,214.355,-82.290,173.794,28.287,155.074
C02908=1070.860,214.106,-82.264,173.792,28.283,155.074
C02909=1070.855,213.858,-82.239,173.790,28.279,155.073
C02910=1070.849,213.609,-82.213,173.788,28.275,155.073
C02911=1070.842,213.360,-82.188,173.786,28.271,155.072
C02912=1070.837,213.111,-82.162,173.784,28.267,155.071
C02913=1070.832,212.863,-82.138,173.781,28.263,155.071
C02914=1070.825,212.614,-82.113,173.780,28.260,155.070
C02915=1070.819,212.365,-82.087,173.778,28.256,155.069
C02916=1070.814,212.116,-82.061,173.775,28.251,155.069
C02917=1070.808,211.868,-82.036,173.774,28.248,155.068
C02918=1070.802,211.620,-82.011,173.772,28.244,155.067
C02919=1070.796,211.370,-81.986,173.769,28.240,155.067
C02920=1070.790,211.122,-81.961,173.768,28.236,155.066
C02921=1070.784,210.874,-81.936,173.765,28.232,155.065
C02922=1070.779,210.625,-81.910,173.763,28.228,155.065
C02923=1070.773,210.376,-81.886,173.761,28.224,155.064
C02924=1070.767,210.127,-81.860,173.759,28.220,155.064
C02925=1070.761,209.879,-81.835,173.757,28.216,155.063
C02926=1070.755,209.630,-81.810,173.755,28.212,155.062
C02927=1070.749,209.381,-81.785,173.753,28.208,155.062
C02928=1070.744,209.170,-81.764,173.752,28.205,155.061
C02929=1070.739,208.958,-81.742,173.749,28.201,155.060
C02930=1070.734,208.745,-81.721,173.748,28.197,155.060
C02931=1070.729,208.533,-81.700,173.746,28.194,155.059
C02932=1070.725,208.321,-81.678,173.744,28.191,155.059
C02933=1070.719,208.109,-81.657,173.742,28.187,155.058
C02934=1070.714,207.897,-81.636,173.741,28.184,155.058
C02935=1070.685,206.642,-81.512,173.603,28.111,155.055
C02936=1070.680,206.393,-81.488,173.601,28.108,155.054
C02937=1070.674,206.145,-81.464,173.599,28.104,155.054
C02938=1070.668,205.896,-81.440,173.596,28.101,155.054
C02939=1070.662,205.648,-81.415,173.594,28.098,155.053
C02940=1070.657,205.399,-81.391,173.592,28.095,155.053
C02941=1070.650,205.150,-81.367,173.590,28.092,155.052
C02942=1070.645,204.901,-81.343,173.587,28.089,155.052
C02943=1070.640,204.652,-81.319,173.586,28.086,155.051
C02944=1070.634,204.403,-81.294,173.583,28.083,155.051
C02945=1070.628,204.155,-81.271,173.581,28.080,155.051
C02946=1070.623,203.906,-81.246,173.578,28.077,155.050
C02947=1070.617,203.657,-81.222,173.577,28.074,155.050
C02948=1070.612,203.408,-81.197,173.574,28.071,155.049
C02949=1070.606,203.160,-81.174,173.572,28.068,155.049
C02950=1070.600,202.911,-81.149,173.570,28.064,155.048
C02951=1070.594,202.662,-81.125,173.568,28.061,155.048
C02952=1070.589,202.413,-81.101,173.565,28.059,155.048
C02953=1070.583,202.165,-81.077,173.564,28.056,155.047
C02954=1070.577,201.915,-81.053,173.561,28.052,155.047
C02955=1070.571,201.667,-81.029,173.559,28.049,155.046
C02956=1070.566,201.418,-81.005,173.556,28.046,155.046
C02957=1070.560,201.169,-80.981,173.555,28.044,155.045
C02958=1070.554,200.921,-80.957,173.552,28.041,155.045
C02959=1070.548,200.672,-80.934,173.550,28.038,155.045
C02960=1070.542,200.423,-80.910,173.548,28.035,155.044
C02961=1070.537,200.174,-80.886,173.546,28.032,155.044
C02962=1070.531,199.926,-80.862,173.543,28.028,155.043
C02963=1070.525,199.676,-80.838,173.542,28.026,155.043
C02964=1070.519,199.428,-80.814,173.539,28.023,155.043
C02965=1070.514,199.179,-80.790,173.537,28.020,155.042
C02966=1070.508,198.930,-80.767,173.535,28.017,155.042
C02967=1070.502,198.681,-80.743,173.533,28.014,155.041
C02968=1070.496,198.433,-80.719,173.530,28.011,155.041
C02969=1070.491,198.184,-80.695,173.529,28.008,155.040
C02970=1070.485,197.935,-80.672,173.526,28.005,155.040
C02971=1070.478,197.686,-80.648,173.524,28.002,155.040
C02972=1070.473,197.437,-80.624,173.522,27.999,155.039
C02973=1070.467,197.189,-80.600,173.520,27.996,155.039
C02974=1070.462,196.940,-80.576,173.517,27.993,155.038
C02975=1070.456,196.691,-80.553,173.516,27.990,155.038
C02976=1070.450,196.442,-80.529,173.513,27.987,155.038
C02977=1070.445,196.193,-80.506,173.511,27.984,155.037
C02978=1070.439,195.945,-80.482,173.509,27.981,155.037
C02979=1070.433,195.696,-80.458,173.507,27.978,155.036
C02980=1070.427,195.447,-80.434,173.504,27.975,155.036
C02981=1070.422,195.198,-80.410,173.503,27.972,155.036
C02982=1070.416,194.949,-80.387,173.500,27.969,155.035
C02983=1070.410,194.701,-80.364,173.499,27.967,155.035
C02984=1070.405,194.452,-80.340,173.496,27.964,155.034
C02985=1070.399,194.204,-80.316,173.494,27.960,155.034
C02986=1070.392,193.954,-80.293,173.492,27.957,155.033
C02987=1070.387,193.705,-80.269,173.490,27.955,155.033
C02988=1070.381,193.456,-80.246,173.487,27.952,155.033
C02989=1070.376,193.208,-80.222,173.486,27.949,155.032
C02990=1070.370,192.959,-80.199,173.483,27.946,155.032
C02991=1070.365,192.710,-80.176,173.482,27.943,155.031
C02992=1070.359,192.462,-80.151,173.479,27.940,155.031
C02993=1070.354,192.213,-80.129,173.477,27.937,155.031
C02994=1070.347,191.964,-80.104,173.475,27.934,155.030
C02995=1070.342,191.714,-80.081,173.473,27.931,155.030
C02996=1070.336,191.433,-80.055,173.470,27.927,155.029
C02997=1070.329,191.151,-80.028,173.468,27.924,155.029
C02998=1070.323,190.869,-80.002,173.465,27.921,155.028
C02999=1070.316,190.587,-79.975,173.463,27.917,155.028
C03000=1070.310,190.338,-79.951,173.461,27.914,155.027
C03001=1070.305,190.089,-79.928,173.459,27.911,155.027
C03002=1070.299,189.840,-79.905,173.457,27.909,155.027
C03003=1070.294,189.591,-79.882,173.455,27.906,155.026
C03004=1070.288,189.343,-79.858,173.453,27.903,155.026
C03005=1070.283,189.094,-79.835,173.451,27.900,155.025
C03006=1070.277,188.845,-79.812,173.448,27.896,155.025
C03007=1070.272,188.596,-79.788,173.447,27.894,155.025
C03008=1070.266,188.347,-79.765,173.444,27.891,155.024
C03009=1070.260,188.099,-79.742,173.443,27.888,155.024
C03010=1070.255,187.849,-79.718,173.440,27.885,155.023
C03011=1070.249,187.600,-79.695,173.439,27.882,155.023
C03012=1070.243,187.352,-79.672,173.436,27.879,155.023
C03013=1070.238,187.103,-79.649,173.434,27.876,155.022
C03014=1070.233,186.854,-79.625,173.432,27.873,155.022
C03015=1070.227,186.605,-79.602,173.430,27.870,155.021
C03016=1070.221,186.356,-79.579,173.428,27.867,155.021
C03017=1070.216,186.107,-79.556,173.426,27.864,155.020
C03018=1070.210,185.859,-79.532,173.424,27.862,155.020
C03019=1070.204,185.610,-79.509,173.422,27.859,155.020
C03020=1070.199,185.361,-79.486,173.420,27.855,155.019
C03021=1070.194,185.113,-79.463,173.418,27.852,155.019
C03022=1070.189,184.864,-79.440,173.416,27.850,155.018
C03023=1070.183,184.615,-79.417,173.414,27.847,155.018
C03024=1070.177,184.365,-79.394,173.411,27.844,155.018
C03025=1070.171,184.116,-79.371,173.410,27.841,155.017
C03026=1070.164,183.868,-79.348,173.407,27.838,155.017
C03027=1070.159,183.619,-79.325,173.406,27.836,155.017
C03028=1070.153,183.370,-79.302,173.403,27.833,155.016
C03029=1070.147,183.121,-79.280,173.402,27.830,155.016
C03030=1070.141,182.872,-79.257,173.399,27.827,155.015
C03031=1070.136,182.623,-79.234,173.398,27.824,155.015
C03032=1070.129,182.375,-79.211,173.395,27.821,155.015
C03033=1070.124,182.126,-79.188,173.394,27.818,155.014
C03034=1070.118,181.877,-79.165,173.391,27.815,155.014
C03035=1070.112,181.628,-79.142,173.389,27.813,155.013
C03036=1070.106,181.379,-79.120,173.387,27.810,155.013
C03037=1070.101,181.130,-79.097,173.385,27.807,155.013
C03038=1070.094,180.882,-79.074,173.383,27.804,155.012
C03039=1070.089,180.632,-79.052,173.381,27.801,155.012
C03040=1070.083,180.383,-79.029,173.379,27.799,155.011
C03041=1070.077,180.134,-79.006,173.377,27.796,155.011
C03042=1070.072,179.885,-78.983,173.375,27.793,155.011
C03043=1070.065,179.637,-78.961,173.373,27.790,155.010
C03044=1070.059,179.388,-78.938,173.371,27.788,155.010
C03045=1070.054,179.139,-78.915,173.368,27.785,155.010
C03046=1070.048,178.889,-78.893,173.367,27.782,155.009
C03047=1070.043,178.641,-78.870,173.364,27.779,155.009
C03048=1070.037,178.393,-78.848,173.363,27.776,155.008
C03049=1070.031,178.144,-78.825,173.360,27.773,155.008
C03050=1070.025,177.895,-78.802,173.359,27.771,155.008
C03051=1070.020,177.645,-78.780,173.356,27.768,155.007
C03052=1070.013,177.397,-78.757,173.355,27.765,155.007
C03053=1070.007,177.148,-78.734,173.352,27.762,155.006
C03054=1070.002,176.898,-78.712,173.351,27.759,155.006
C03055=1069.996,176.649,-78.689,173.348,27.757,155.006
C03056=1069.990,176.401,-78.667,173.347,27.754,155.005
C03057=1069.985,176.153,-78.644,173.344,27.751,155.005
C03058=1069.979,175.903,-78.622,173.343,27.748,155.005
C03059=1069.974,175.654,-78.599,173.340,27.745,155.004
C03060=1069.967,175.372,-78.574,173.339,27.742,155.004
C03061=1069.960,175.089,-78.548,173.336,27.739,155.003
C03062=1069.953,174.807,-78.523,173.334,27.736,155.003
C03063=1069.948,174.525,-78.497,173.332,27.732,155.002
C03064=1069.941,174.276,-78.475,173.330,27.729,155.002
C03065=1069.935,174.027,-78.452,173.328,27.726,155.002
C03066=1069.930,173.778,-78.430,173.326,27.724,155.001
C03067=1069.925,173.529,-78.407,173.324,27.721,155.001
C03068=1069.919,173.280,-78.385,173.322,27.718,155.001
C03069=1069.913,173.031,-78.363,173.320,27.716,155.000
C03070=1069.907,172.782,-78.340,173.318,27.713,155.000
C03071=1069.902,172.534,-78.318,173.316,27.710,154.999
C03072=1069.896,172.285,-78.295,173.314,27.707,154.999
C03073=1069.890,172.035,-78.273,173.312,27.704,154.999
C03074=1069.885,171.787,-78.250,173.310,27.701,154.998
C03075=1069.879,171.538,-78.229,173.308,27.698,154.998
C03076=1069.873,171.289,-78.206,173.306,27.695,154.997
C03077=1069.868,171.040,-78.184,173.304,27.693,154.997
C03078=1069.861,170.791,-78.161,173.303,27.690,154.997
C03079=1069.857,170.542,-78.140,173.300,27.687,154.996
C03080=1069.851,170.293,-78.117,173.299,27.684,154.996
C03081=1069.845,170.044,-78.095,173.296,27.681,154.995
C03082=1069.839,169.795,-78.072,173.295,27.678,154.995
C03083=1069.834,169.546,-78.050,173.292,27.675,154.995
C03084=1069.828,169.297,-78.029,173.291,27.673,154.994
C03085=1069.822,169.048,-78.006,173.289,27.670,154.994
C03086=1069.817,168.799,-77.983,173.287,27.667,154.993
C03087=1069.811,168.551,-77.961,173.285,27.664,154.993
C03088=1069.806,168.301,-77.939,173.283,27.662,154.993
C03089=1069.800,168.052,-77.917,173.281,27.659,154.992
C03090=1069.794,167.804,-77.895,173.279,27.656,154.992
C03091=1069.789,167.554,-77.873,173.277,27.653,154.991
C03092=1069.783,167.306,-77.850,173.276,27.650,154.991
C03093=1069.778,167.057,-77.828,173.273,27.647,154.991
C03094=1069.772,166.808,-77.806,173.272,27.645,154.990
C03095=1069.766,166.559,-77.784,173.269,27.642,154.990
C03096=1069.761,166.310,-77.762,173.268,27.639,154.990
C03097=1069.755,166.061,-77.740,173.266,27.636,154.989
C03098=1069.750,165.812,-77.719,173.264,27.633,154.989
C03099=1069.744,165.563,-77.696,173.262,27.630,154.988
C03100=1069.739,165.314,-77.673,173.261,27.627,154.988
C03101=1069.733,165.065,-77.652,173.258,27.624,154.988
C03102=1069.728,164.816,-77.630,173.257,27.622,154.987
C03103=1069.721,164.567,-77.607,173.254,27.619,154.987
C03104=1069.716,164.318,-77.586,173.253,27.616,154.986
C03105=1069.711,164.069,-77.563,173.251,27.613,154.986
C03106=1069.705,163.820,-77.542,173.249,27.610,154.986
C03107=1069.700,163.571,-77.519,173.247,27.607,154.985
C03108=1069.694,163.323,-77.498,173.245,27.604,154.985
C03109=1069.689,163.073,-77.476,173.243,27.602,154.984
C03110=1069.683,162.824,-77.453,173.242,27.599,154.984
C03111=1069.678,162.575,-77.432,173.239,27.596,154.984
C03112=1069.672,162.326,-77.410,173.238,27.593,154.983
C03113=1069.666,162.078,-77.388,173.236,27.590,154.983
C03114=1069.661,161.828,-77.366,173.234,27.587,154.982
C03115=1069.655,161.580,-77.344,173.232,27.584,154.982
C03116=1069.650,161.330,-77.322,173.231,27.582,154.982
C03117=1069.644,161.081,-77.301,173.229,27.579,154.981
C03118=1069.639,160.832,-77.279,173.227,27.576,154.981
C03119=1069.633,160.583,-77.257,173.225,27.573,154.980
C03120=1069.627,160.335,-77.236,173.223,27.570,154.980
C03121=1069.621,160.085,-77.214,173.222,27.567,154.980
C03122=1069.616,159.836,-77.192,173.219,27.565,154.979
C03123=1069.610,159.587,-77.171,173.217,27.562,154.979
C03124=1069.603,159.305,-77.146,173.215,27.559,154.978
C03125=1069.597,159.023,-77.121,173.214,27.556,154.978
C03126=1069.590,158.739,-77.097,173.211,27.553,154.978
C03127=1069.584,158.457,-77.072,173.209,27.549,154.977
C03128=1069.578,158.208,-77.051,173.207,27.546,154.977
C03129=1069.573,157.958,-77.029,173.206,27.544,154.976
C03130=1069.567,157.710,-77.007,173.203,27.541,154.976
C03131=1069.561,157.461,-76.986,173.202,27.538,154.976
C03132=1069.555,157.212,-76.965,173.200,27.536,154.975
C03133=1069.550,156.963,-76.942,173.198,27.533,154.975
C03134=1069.544,156.714,-76.921,173.196,27.530,154.974
C03135=1069.538,156.465,-76.899,173.195,27.527,154.974
C03136=1069.532,156.216,-76.878,173.192,27.525,154.974
C03137=1069.527,155.967,-76.857,173.191,27.522,154.973
C03138=1069.521,155.717,-76.835,173.189,27.519,154.973
C03139=1069.516,155.469,-76.814,173.187,27.516,154.973
C03140=1069.510,155.219,-76.792,173.185,27.513,154.972
C03141=1069.504,154.971,-76.771,173.184,27.510,154.972
C03142=1069.498,154.722,-76.749,173.181,27.508,154.971
C03143=1069.492,154.473,-76.728,173.180,27.505,154.971
C03144=1069.486,154.223,-76.707,173.178,27.502,154.971
C03145=1069.482,153.975,-76.685,173.176,27.499,154.970
C03146=1069.475,153.725,-76.663,173.174,27.497,154.970
C03147=1069.470,153.477,-76.642,173.173,27.494,154.969
C03148=1069.464,153.227,-76.621,173.170,27.491,154.969
C03149=1069.458,152.979,-76.600,173.169,27.489,154.969
C03150=1069.452,152.729,-76.578,173.167,27.486,154.968
C03151=1069.447,152.481,-76.557,173.165,27.483,154.968
C03152=1069.441,152.231,-76.536,173.163,27.480,154.968
C03153=1069.435,151.983,-76.515,173.162,27.477,154.967
C03154=1069.429,151.733,-76.493,173.159,27.475,154.967
C03155=1069.424,151.485,-76.472,173.158,27.472,154.967
C03156=1069.418,151.235,-76.451,173.156,27.469,154.966
C03157=1069.412,150.987,-76.430,173.155,27.467,154.966
C03158=1069.406,150.737,-76.408,173.152,27.463,154.965
C03159=1069.402,150.488,-76.387,173.151,27.461,154.965
C03160=1069.396,150.239,-76.366,173.149,27.458,154.965
C03161=1069.390,149.990,-76.344,173.147,27.455,154.964
C03162=1069.385,149.741,-76.324,173.145,27.453,154.964
C03163=1069.378,149.492,-76.302,173.144,27.450,154.963
C03164=1069.373,149.243,-76.281,173.142,27.447,154.963
C03165=1069.367,148.994,-76.260,173.140,27.444,154.963
C03166=1069.361,148.745,-76.239,173.138,27.441,154.962
C03167=1069.356,148.496,-76.218,173.137,27.439,154.962
C03168=1069.349,148.247,-76.197,173.134,27.436,154.962
C03169=1069.344,147.998,-76.176,173.133,27.433,154.961
C03170=1069.338,147.749,-76.155,173.131,27.431,154.961
C03171=1069.332,147.500,-76.133,173.130,27.428,154.960
C03172=1069.326,147.250,-76.113,173.127,27.425,154.960
C03173=1069.321,147.002,-76.091,173.126,27.422,154.960
C03174=1069.316,146.753,-76.071,173.124,27.420,154.959
C03175=1069.309,146.503,-76.049,173.122,27.417,154.959
C03176=1069.303,146.255,-76.029,173.120,27.414,154.958
C03177=1069.297,146.005,-76.007,173.119,27.412,154.958
C03178=1069.292,145.756,-75.987,173.117,27.409,154.958
C03179=1069.286,145.508,-75.966,173.115,27.406,154.957
C03180=1069.281,145.258,-75.945,173.113,27.403,154.957
C03181=1069.275,145.010,-75.923,173.112,27.400,154.957
C03182=1069.268,144.760,-75.903,173.110,27.398,154.956
C03183=1069.263,144.512,-75.882,173.108,27.395,154.956
C03184=1069.258,144.262,-75.861,173.106,27.392,154.956
C03185=1069.252,144.013,-75.840,173.105,27.389,154.955
C03186=1069.246,143.764,-75.819,173.102,27.386,154.955
C03187=1069.240,143.515,-75.799,173.101,27.384,154.954
C03188=1069.234,143.233,-75.775,173.099,27.381,154.954
C03189=1069.228,142.949,-75.751,173.097,27.378,154.954
C03190=1069.221,142.666,-75.728,173.095,27.374,154.953
C03191=1069.214,142.383,-75.704,173.093,27.371,154.953
C03192=1069.209,142.134,-75.683,173.091,27.369,154.952
C03193=1069.203,141.884,-75.662,173.090,27.366,154.952
C03194=1069.197,141.636,-75.642,173.087,27.363,154.952
C03195=1069.192,141.387,-75.621,173.086,27.361,154.951
C03196=1069.186,141.137,-75.600,173.084,27.358,154.951
C03197=1069.180,140.889,-75.579,173.083,27.355,154.950
C03198=1069.174,140.640,-75.559,173.080,27.352,154.950
C03199=1069.168,140.390,-75.538,173.079,27.349,154.950
C03200=1069.163,140.142,-75.517,173.077,27.347,154.949
C03201=1069.158,139.893,-75.496,173.076,27.344,154.949
C03202=1069.151,139.643,-75.476,173.073,27.341,154.949
C03203=1069.146,139.394,-75.455,173.072,27.338,154.948
C03204=1069.141,139.145,-75.435,173.071,27.336,154.948
C03205=1069.134,138.897,-75.414,173.069,27.333,154.947
C03206=1069.128,138.647,-75.393,173.066,27.330,154.947
C03207=1069.122,138.398,-75.373,173.065,27.328,154.947
C03208=1069.117,138.149,-75.353,173.064,27.325,154.946
C03209=1069.111,137.900,-75.331,173.062,27.322,154.946
C03210=1069.105,137.651,-75.311,173.060,27.320,154.946
C03211=1069.100,137.402,-75.291,173.058,27.317,154.945
C03212=1069.094,137.153,-75.271,173.057,27.314,154.945
C03213=1069.088,136.903,-75.250,173.055,27.311,154.944
C03214=1069.083,136.654,-75.229,173.054,27.308,154.944
C03215=1069.077,136.405,-75.209,173.051,27.306,154.944
C03216=1069.071,136.157,-75.188,173.050,27.303,154.943
C03217=1069.064,135.907,-75.168,173.048,27.300,154.943
C03218=1069.059,135.658,-75.147,173.047,27.297,154.942
C03219=1069.053,135.409,-75.127,173.045,27.295,154.942
C03220=1069.048,135.160,-75.106,173.043,27.292,154.942
C03221=1069.042,134.910,-75.086,173.041,27.289,154.941
C03222=1069.036,134.661,-75.066,173.040,27.287,154.941
C03223=1069.031,134.412,-75.045,173.038,27.284,154.941
C03224=1069.025,134.163,-75.025,173.037,27.281,154.940
C03225=1069.019,133.914,-75.004,173.034,27.279,154.940
C03226=1069.013,133.665,-74.984,173.033,27.276,154.940
C03227=1069.008,133.416,-74.964,173.031,27.273,154.939
C03228=1069.002,133.167,-74.944,173.030,27.270,154.939
C03229=1068.996,132.918,-74.923,173.028,27.267,154.938
C03230=1068.990,132.669,-74.903,173.026,27.264,154.938
C03231=1068.985,132.419,-74.882,173.024,27.262,154.938
C03232=1068.979,132.170,-74.862,173.023,27.259,154.937
C03233=1068.973,131.921,-74.842,173.021,27.257,154.937
C03234=1068.967,131.672,-74.822,173.020,27.254,154.936
C03235=1068.962,131.423,-74.801,173.017,27.251,154.936
C03236=1068.956,131.174,-74.781,173.016,27.248,154.936
C03237=1068.950,130.925,-74.761,173.014,27.246,154.935
C03238=1068.944,130.676,-74.741,173.013,27.243,154.935
C03239=1068.938,130.427,-74.720,173.011,27.241,154.935
C03240=1068.932,130.177,-74.700,173.009,27.238,154.934
C03241=1068.926,129.929,-74.680,173.007,27.235,154.934
C03242=1068.921,129.679,-74.660,173.006,27.233,154.934
C03243=1068.915,129.430,-74.640,173.004,27.230,154.933
C03244=1068.909,129.181,-74.620,173.003,27.227,154.933
C03245=1068.902,128.932,-74.600,173.000,27.224,154.932
C03246=1068.897,128.683,-74.580,172.999,27.222,154.932
C03247=1068.891,128.434,-74.560,172.997,27.219,154.932
C03248=1068.885,128.184,-74.540,172.996,27.216,154.931
C03249=1068.879,127.936,-74.520,172.994,27.213,154.931
C03250=1068.874,127.686,-74.500,172.993,27.211,154.931
C03251=1068.867,127.437,-74.479,172.990,27.208,154.930
C03252=1068.861,127.155,-74.457,172.989,27.205,154.930
C03253=1068.855,126.871,-74.434,172.986,27.202,154.929
C03254=1068.848,126.588,-74.411,172.985,27.199,154.929
C03255=1068.841,126.304,-74.389,172.983,27.196,154.929
C03256=1068.835,126.056,-74.369,172.981,27.193,154.928
C03257=1068.829,125.807,-74.349,172.980,27.190,154.928
C03258=1068.824,125.558,-74.329,172.978,27.188,154.927
C03259=1068.818,125.308,-74.309,172.977,27.185,154.927
C03260=1068.812,125.059,-74.289,172.975,27.182,154.927
C03261=1068.806,124.811,-74.269,172.974,27.179,154.926
C03262=1068.800,124.562,-74.250,172.971,27.176,154.926
C03263=1068.795,124.311,-74.229,172.970,27.174,154.926
C03264=1068.789,124.062,-74.209,172.968,27.171,154.925
C03265=1068.783,123.814,-74.189,172.967,27.169,154.925
C03266=1068.777,123.564,-74.170,172.965,27.166,154.924
C03267=1068.772,123.315,-74.150,172.964,27.163,154.924
C03268=1068.766,123.066,-74.130,172.961,27.160,154.924
C03269=1068.760,122.817,-74.110,172.960,27.158,154.923
C03270=1068.754,122.568,-74.090,172.958,27.155,154.923
C03271=1068.748,122.319,-74.071,172.957,27.152,154.923
C03272=1068.742,122.070,-74.051,172.955,27.149,154.922
C03273=1068.737,121.821,-74.031,172.954,27.147,154.922
C03274=1068.731,121.571,-74.011,172.952,27.144,154.921
C03275=1068.725,121.322,-73.991,172.950,27.141,154.921
C03276=1068.720,121.073,-73.972,172.948,27.138,154.921
C03277=1068.714,120.824,-73.952,172.947,27.136,154.920
C03278=1068.709,120.574,-73.932,172.945,27.133,154.920
C03279=1068.703,120.326,-73.912,172.944,27.131,154.920
C03280=1068.697,120.077,-73.893,172.942,27.128,154.919
C03281=1068.691,119.827,-73.873,172.941,27.125,154.919
C03282=1068.685,119.579,-73.853,172.939,27.122,154.918
C03283=1068.680,119.329,-73.834,172.937,27.119,154.918
C03284=1068.674,119.080,-73.814,172.936,27.116,154.918
C03285=1068.669,118.831,-73.794,172.934,27.114,154.917
C03286=1068.663,118.582,-73.774,172.932,27.111,154.917
C03287=1068.657,118.332,-73.755,172.931,27.108,154.916
C03288=1068.651,118.083,-73.736,172.930,27.106,154.916
C03289=1068.645,117.834,-73.716,172.928,27.103,154.916
C03290=1068.640,117.585,-73.697,172.926,27.100,154.915
C03291=1068.634,117.336,-73.676,172.924,27.097,154.915
C03292=1068.629,117.086,-73.657,172.923,27.095,154.915
C03293=1068.623,116.837,-73.637,172.921,27.092,154.914
C03294=1068.617,116.588,-73.618,172.920,27.089,154.914
C03295=1068.611,116.339,-73.598,172.918,27.086,154.913
C03296=1068.605,116.090,-73.578,172.917,27.084,154.913
C03297=1068.600,115.840,-73.559,172.915,27.081,154.913
C03298=1068.594,115.592,-73.540,172.914,27.078,154.912
C03299=1068.589,115.342,-73.520,172.911,27.075,154.912
C03300=1068.583,115.093,-73.500,172.910,27.072,154.911
C03301=1068.577,114.844,-73.481,172.908,27.070,154.911
C03302=1068.572,114.595,-73.461,172.907,27.067,154.911
C03303=1068.566,114.345,-73.442,172.905,27.064,154.910
C03304=1068.560,114.096,-73.422,172.904,27.061,154.910
C03305=1068.554,113.847,-73.403,172.903,27.059,154.909
C03306=1068.549,113.598,-73.384,172.901,27.056,154.909
C03307=1068.543,113.349,-73.364,172.899,27.054,154.909
C03308=1068.537,113.099,-73.344,172.897,27.050,154.908
C03309=1068.531,112.850,-73.325,172.896,27.048,154.908
C03310=1068.526,112.601,-73.307,172.894,27.045,154.908
C03311=1068.520,112.353,-73.287,172.893,27.042,154.907
C03312=1068.514,112.103,-73.268,172.891,27.040,154.907
C03313=1068.508,111.854,-73.248,172.890,27.037,154.907
C03314=1068.502,111.604,-73.229,172.888,27.034,154.906
C03315=1068.497,111.355,-73.209,172.887,27.031,154.906
C03316=1068.488,110.979,-73.180,172.885,27.027,154.905
C03317=1068.478,110.601,-73.151,172.881,27.023,154.905
C03318=1068.470,110.225,-73.122,172.879,27.019,154.904
C03319=1068.461,109.847,-73.094,172.877,27.015,154.903
C03320=1068.455,109.598,-73.074,172.875,27.013,154.903
C03321=1068.449,109.349,-73.055,172.874,27.010,154.903
C03322=1068.443,109.100,-73.036,172.872,27.007,154.902
C03323=1068.438,108.850,-73.017,172.871,27.004,154.902
C03324=1068.432,108.601,-72.997,172.870,27.001,154.902
C03325=1068.425,108.352,-72.979,172.867,26.999,154.901
C03326=1068.420,108.102,-72.959,172.866,26.996,154.901
C03327=1068.415,107.854,-72.941,172.864,26.993,154.901
C03328=1068.409,107.605,-72.921,172.863,26.990,154.900
C03329=1068.402,107.356,-72.902,172.861,26.988,154.900
C03330=1068.397,107.106,-72.883,172.860,26.985,154.899
C03331=1068.391,106.857,-72.863,172.858,26.982,154.899
C03332=1068.385,106.607,-72.844,172.857,26.980,154.899
C03333=1068.379,106.358,-72.826,172.855,26.977,154.898
C03334=1068.374,106.110,-72.807,172.854,26.975,154.898
C03335=1068.368,105.860,-72.787,172.852,26.972,154.898
C03336=1068.362,105.611,-72.769,172.851,26.969,154.897
C03337=1068.356,105.362,-72.750,172.848,26.966,154.897
C03338=1068.350,105.112,-72.730,172.847,26.963,154.896
C03339=1068.345,104.863,-72.711,172.845,26.960,154.896
C03340=1068.339,104.614,-72.693,172.844,26.958,154.896
C03341=1068.333,104.365,-72.674,172.842,26.955,154.895
C03342=1068.327,104.115,-72.654,172.841,26.952,154.895
C03343=1068.321,103.866,-72.636,172.840,26.950,154.894
C03344=1068.316,103.618,-72.617,172.838,26.947,154.894
C03345=1068.310,103.368,-72.598,172.837,26.944,154.894
C03346=1068.304,103.119,-72.579,172.835,26.942,154.893
C03347=1068.298,102.870,-72.560,172.834,26.939,154.893
C03348=1068.293,102.621,-72.541,172.832,26.936,154.893
C03349=1068.288,102.371,-72.522,172.831,26.933,154.892
C03350=1068.281,102.122,-72.504,172.828,26.930,154.892
C03351=1068.275,101.872,-72.484,172.827,26.927,154.891
C03352=1068.266,101.468,-72.454,172.825,26.923,154.891
C03353=1068.257,101.064,-72.423,172.822,26.919,154.890
C03354=1068.247,100.659,-72.393,172.819,26.914,154.890
C03355=1068.238,100.254,-72.362,172.817,26.910,154.889
C03356=1068.231,100.005,-72.343,172.816,26.907,154.889
C03357=1068.226,99.756,-72.326,172.814,26.905,154.888
C03358=1068.220,99.507,-72.306,172.813,26.902,154.888
C03359=1068.214,99.258,-72.288,172.811,26.899,154.888
C03360=1068.208,99.008,-72.268,172.810,26.897,154.887
C03361=1068.202,98.759,-72.250,172.808,26.894,154.887
C03362=1068.197,98.510,-72.232,172.807,26.891,154.886
C03363=1068.190,98.261,-72.213,172.805,26.889,154.886
C03364=1068.185,98.011,-72.194,172.803,26.886,154.886
C03365=1068.178,97.762,-72.175,172.802,26.883,154.885
C03366=1068.174,97.513,-72.157,172.800,26.880,154.885
C03367=1068.167,97.264,-72.138,172.799,26.877,154.884
C03368=1068.161,97.014,-72.120,172.797,26.875,154.884
C03369=1068.156,96.766,-72.101,172.796,26.872,154.884
C03370=1068.150,96.516,-72.083,172.794,26.869,154.883
C03371=1068.144,96.266,-72.064,172.793,26.866,154.883
C03372=1068.137,96.017,-72.045,172.791,26.864,154.883
C03373=1068.133,95.768,-72.027,172.790,26.861,154.882
C03374=1068.126,95.519,-72.008,172.788,26.859,154.882
C03375=1068.120,95.270,-71.989,172.787,26.856,154.881
C03376=1068.113,94.987,-71.969,172.785,26.853,154.881
C03377=1068.107,94.704,-71.947,172.783,26.849,154.881
C03378=1068.101,94.420,-71.926,172.782,26.846,154.880
C03379=1068.095,94.137,-71.906,172.780,26.844,154.880
C03380=1068.088,93.888,-71.887,172.779,26.841,154.879
C03381=1068.082,93.639,-71.868,172.777,26.838,154.879
C03382=1068.077,93.389,-71.850,172.775,26.835,154.879
C03383=1068.071,93.140,-71.831,172.774,26.832,154.878
C03384=1068.065,92.890,-71.813,172.772,26.829,154.878
C03385=1068.059,92.642,-71.795,172.771,26.827,154.878
C03386=1068.053,92.393,-71.776,172.769,26.824,154.877
C03387=1068.048,92.143,-71.758,172.768,26.821,154.877
C03388=1068.042,91.894,-71.739,172.766,26.818,154.876
C03389=1068.036,91.644,-71.721,172.765,26.816,154.876
C03390=1068.031,91.396,-71.702,172.763,26.813,154.876
C03391=1068.024,91.146,-71.684,172.762,26.810,154.875
C03392=1068.019,90.897,-71.665,172.760,26.808,154.875
C03393=1068.013,90.648,-71.648,172.759,26.805,154.874
C03394=1068.007,90.398,-71.629,172.757,26.802,154.874
C03395=1068.001,90.149,-71.611,172.756,26.799,154.874
C03396=1067.995,89.900,-71.593,172.754,26.797,154.873
C03397=1067.990,89.650,-71.574,172.753,26.794,154.873
C03398=1067.984,89.402,-71.556,172.752,26.791,154.873
C03399=1067.978,89.152,-71.538,172.750,26.789,154.872
C03400=1067.971,88.902,-71.520,172.749,26.786,154.872
C03401=1067.966,88.654,-71.502,172.747,26.783,154.871
C03402=1067.959,88.404,-71.484,172.746,26.781,154.871
C03403=1067.954,88.155,-71.465,172.744,26.778,154.871
C03404=1067.948,87.906,-71.447,172.743,26.776,154.870
C03405=1067.942,87.657,-71.428,172.741,26.773,154.870
C03406=1067.936,87.408,-71.411,172.740,26.770,154.870
C03407=1067.930,87.158,-71.393,172.738,26.767,154.869
C03408=1067.924,86.909,-71.374,172.737,26.764,154.869
C03409=1067.918,86.660,-71.357,172.735,26.762,154.868
C03410=1067.913,86.410,-71.338,172.734,26.759,154.868
C03411=1067.907,86.161,-71.320,172.733,26.756,154.868
C03412=1067.901,85.911,-71.302,172.731,26.753,154.867
C03413=1067.895,85.662,-71.284,172.729,26.751,154.867
C03414=1067.889,85.413,-71.266,172.727,26.748,154.867
C03415=1067.883,85.164,-71.248,172.726,26.745,154.866
C03416=1067.877,84.914,-71.230,172.724,26.742,154.866
C03417=1067.871,84.665,-71.212,172.723,26.740,154.865
C03418=1067.866,84.416,-71.193,172.721,26.737,154.865
C03419=1067.860,84.166,-71.176,172.720,26.735,154.865
C03420=1067.854,83.918,-71.157,172.718,26.732,154.864
C03421=1067.848,83.668,-71.139,172.717,26.729,154.864
C03422=1067.842,83.418,-71.121,172.716,26.726,154.864
C03423=1067.836,83.169,-71.104,172.714,26.724,154.863
C03424=1067.830,82.920,-71.085,172.713,26.721,154.863
C03425=1067.825,82.671,-71.068,172.711,26.718,154.862
C03426=1067.818,82.421,-71.050,172.710,26.715,154.862
C03427=1067.813,82.172,-71.032,172.708,26.712,154.862
C03428=1067.807,81.922,-71.014,172.707,26.710,154.861
C03429=1067.802,81.674,-70.995,172.705,26.707,154.861
C03430=1067.796,81.424,-70.977,172.704,26.704,154.861
C03431=1067.790,81.175,-70.960,172.702,26.702,154.860
C03432=1067.784,80.925,-70.942,172.701,26.699,154.860
C03433=1067.778,80.676,-70.924,172.700,26.696,154.859
C03434=1067.773,80.428,-70.906,172.698,26.693,154.859
C03435=1067.766,80.178,-70.888,172.697,26.690,154.859
C03436=1067.761,79.929,-70.871,172.695,26.688,154.858
C03437=1067.755,79.679,-70.853,172.694,26.685,154.858
C03438=1067.749,79.430,-70.835,172.692,26.682,154.857
C03439=1067.743,79.181,-70.817,172.691,26.680,154.857
C03440=1067.737,78.897,-70.796,172.689,26.677,154.857
C03441=1067.730,78.614,-70.776,172.688,26.673,154.856
C03442=1067.724,78.332,-70.756,172.686,26.670,154.856
C03443=1067.717,78.049,-70.736,172.684,26.667,154.855
C03444=1067.711,77.799,-70.718,172.683,26.665,154.855
C03445=1067.705,77.550,-70.701,172.681,26.662,154.855
C03446=1067.699,77.300,-70.683,172.680,26.659,154.854
C03447=1067.693,77.051,-70.665,172.679,26.657,154.854
C03448=1067.687,76.802,-70.647,172.677,26.654,154.854
C03449=1067.682,76.553,-70.630,172.676,26.651,154.853
C03450=1067.675,76.303,-70.612,172.674,26.648,154.853
C03451=1067.669,76.054,-70.595,172.673,26.646,154.852
C03452=1067.664,75.805,-70.577,172.671,26.643,154.852
C03453=1067.658,75.555,-70.559,172.670,26.640,154.852
C03454=1067.652,75.306,-70.542,172.668,26.637,154.851
C03455=1067.646,75.057,-70.524,172.667,26.635,154.851
C03456=1067.640,74.808,-70.507,172.665,26.632,154.851
C03457=1067.634,74.558,-70.489,172.664,26.629,154.850
C03458=1067.628,74.309,-70.471,172.663,26.626,154.850
C03459=1067.623,74.060,-70.454,172.661,26.624,154.849
C03460=1067.617,73.810,-70.436,172.660,26.621,154.849
C03461=1067.611,73.561,-70.418,172.658,26.619,154.849
C03462=1067.604,73.312,-70.401,172.657,26.616,154.848
C03463=1067.599,73.063,-70.383,172.655,26.613,154.848
C03464=1067.594,72.813,-70.366,172.654,26.610,154.847
C03465=1067.587,72.563,-70.348,172.652,26.608,154.847
C03466=1067.582,72.314,-70.331,172.651,26.605,154.847
C03467=1067.575,72.065,-70.313,172.650,26.602,154.846
C03468=1067.570,71.816,-70.296,172.648,26.599,154.846
C03469=1067.564,71.567,-70.278,172.647,26.596,154.846
C03470=1067.558,71.317,-70.260,172.645,26.594,154.845
C03471=1067.552,71.068,-70.243,172.644,26.591,154.845
C03472=1067.546,70.818,-70.226,172.642,26.588,154.845
C03473=1067.540,70.569,-70.209,172.641,26.586,154.844
C03474=1067.535,70.320,-70.191,172.640,26.583,154.844
C03475=1067.529,70.070,-70.173,172.638,26.580,154.843
C03476=1067.522,69.821,-70.156,172.637,26.578,154.843
C03477=1067.517,69.572,-70.139,172.635,26.575,154.843
C03478=1067.511,69.322,-70.121,172.634,26.572,154.842
C03479=1067.505,69.073,-70.104,172.632,26.569,154.842
C03480=1067.499,68.824,-70.087,172.631,26.567,154.842
C03481=1067.493,68.575,-70.069,172.629,26.564,154.841
C03482=1067.487,68.325,-70.053,172.628,26.561,154.841
C03483=1067.482,68.076,-70.035,172.626,26.558,154.840
C03484=1067.476,67.826,-70.017,172.625,26.556,154.840
C03485=1067.469,67.578,-70.000,172.624,26.553,154.840
C03486=1067.464,67.328,-69.983,172.622,26.550,154.839
C03487=1067.458,67.078,-69.965,172.621,26.547,154.839
C03488=1067.452,66.830,-69.948,172.619,26.545,154.839
C03489=1067.447,66.580,-69.932,172.618,26.542,154.838
C03490=1067.440,66.330,-69.914,172.616,26.540,154.838
C03491=1067.434,66.081,-69.897,172.615,26.537,154.837
C03492=1067.429,65.832,-69.880,172.614,26.534,154.837
C03493=1067.422,65.582,-69.863,172.612,26.532,154.837
C03494=1067.417,65.333,-69.845,172.611,26.529,154.836
C03495=1067.411,65.084,-69.829,172.609,26.526,154.836
C03496=1067.404,64.834,-69.811,172.608,26.523,154.836
C03497=1067.398,64.585,-69.794,172.606,26.521,154.835
C03498=1067.393,64.336,-69.777,172.605,26.518,154.835
C03499=1067.386,64.086,-69.760,172.603,26.515,154.834
C03500=1067.381,63.837,-69.742,172.602,26.513,154.834
C03501=1067.375,63.588,-69.726,172.600,26.510,154.834
C03502=1067.369,63.338,-69.708,172.599,26.507,154.833
C03503=1067.363,63.089,-69.692,172.597,26.505,154.833
C03504=1067.356,62.806,-69.672,172.596,26.501,154.833
C03505=1067.349,62.522,-69.652,172.595,26.498,154.832
C03506=1067.342,62.240,-69.634,172.593,26.496,154.832
C03507=1067.335,61.956,-69.614,172.591,26.493,154.831
C03508=1067.329,61.707,-69.597,172.590,26.490,154.831
C03509=1067.323,61.457,-69.580,172.588,26.487,154.831
C03510=1067.317,61.208,-69.563,172.587,26.485,154.830
C03511=1067.311,60.959,-69.546,172.585,26.482,154.830
C03512=1067.305,60.709,-69.529,172.585,26.479,154.830
C03513=1067.299,60.460,-69.513,172.583,26.477,154.829
C03514=1067.293,60.211,-69.495,172.582,26.474,154.829
C03515=1067.287,59.962,-69.479,172.580,26.471,154.828
C03516=1067.280,59.712,-69.462,172.579,26.469,154.828
C03517=1067.275,59.463,-69.445,172.577,26.466,154.828
C03518=1067.269,59.214,-69.428,172.576,26.463,154.827
C03519=1067.263,58.964,-69.412,172.575,26.461,154.827
C03520=1067.257,58.714,-69.394,172.573,26.458,154.827
C03521=1067.251,58.465,-69.377,172.572,26.455,154.826
C03522=1067.245,58.216,-69.361,172.570,26.453,154.826
C03523=1067.239,57.967,-69.344,172.569,26.450,154.826
C03524=1067.233,57.717,-69.327,172.567,26.447,154.825
C03525=1067.226,57.468,-69.310,172.566,26.444,154.825
C03526=1067.221,57.219,-69.293,172.564,26.442,154.825
C03527=1067.215,56.969,-69.277,172.563,26.439,154.824
C03528=1067.208,56.720,-69.260,172.562,26.436,154.824
C03529=1067.203,56.470,-69.243,172.560,26.434,154.823
C03530=1067.197,56.221,-69.226,172.559,26.431,154.823
C03531=1067.191,55.972,-69.209,172.557,26.428,154.823
C03532=1067.186,55.722,-69.193,172.556,26.425,154.822
C03533=1067.179,55.472,-69.176,172.554,26.423,154.822
C03534=1067.173,55.224,-69.159,172.553,26.420,154.822
C03535=1067.167,54.974,-69.143,172.552,26.417,154.821
C03536=1067.162,54.725,-69.126,172.550,26.415,154.821
C03537=1067.156,54.476,-69.109,172.549,26.412,154.821
C03538=1067.150,54.227,-69.093,172.547,26.409,154.820
C03539=1067.144,53.976,-69.075,172.546,26.407,154.820
C03540=1067.138,53.727,-69.059,172.544,26.404,154.819
C03541=1067.132,53.478,-69.042,172.543,26.401,154.819
C03542=1067.126,53.229,-69.026,172.541,26.399,154.819
C03543=1067.120,52.979,-69.009,172.540,26.396,154.818
C03544=1067.114,52.730,-68.992,172.539,26.393,154.818
C03545=1067.108,52.481,-68.976,172.537,26.391,154.818
C03546=1067.102,52.231,-68.959,172.536,26.388,154.817
C03547=1067.096,51.981,-68.942,172.534,26.385,154.817
C03548=1067.090,51.733,-68.925,172.533,26.383,154.817
C03549=1067.084,51.483,-68.909,172.531,26.380,154.816
C03550=1067.079,51.234,-68.892,172.530,26.377,154.816
C03551=1067.073,50.984,-68.876,172.529,26.374,154.815
C03552=1067.067,50.735,-68.860,172.528,26.372,154.815
C03553=1067.061,50.486,-68.843,172.527,26.369,154.815
C03554=1067.055,50.237,-68.827,172.525,26.366,154.814
C03555=1067.049,49.986,-68.809,172.524,26.363,154.814
C03556=1067.043,49.737,-68.793,172.522,26.361,154.814
C03557=1067.037,49.488,-68.777,172.521,26.358,154.813
C03558=1067.031,49.238,-68.761,172.519,26.355,154.813
C03559=1067.026,48.989,-68.744,172.518,26.353,154.812
C03560=1067.020,48.740,-68.727,172.517,26.350,154.812
C03561=1067.014,48.491,-68.711,172.515,26.347,154.812
C03562=1067.008,48.241,-68.694,172.514,26.345,154.811
C03563=1067.003,47.992,-68.677,172.512,26.342,154.811
C03564=1066.997,47.742,-68.661,172.511,26.339,154.810
C03565=1066.991,47.493,-68.645,172.509,26.337,154.810
C03566=1066.985,47.244,-68.629,172.508,26.334,154.810
C03567=1066.979,46.994,-68.612,172.507,26.331,154.809
C03568=1066.972,46.711,-68.593,172.505,26.328,154.809
C03569=1066.966,46.427,-68.575,172.504,26.325,154.809
C03570=1066.959,46.144,-68.556,172.502,26.321,154.808
C03571=1066.953,45.860,-68.538,172.500,26.319,154.808
C03572=1066.947,45.611,-68.522,172.499,26.316,154.807
C03573=1066.942,45.361,-68.505,172.497,26.313,154.807
C03574=1066.936,45.112,-68.488,172.496,26.311,154.807
C03575=1066.930,44.863,-68.472,172.495,26.308,154.806
C03576=1066.924,44.613,-68.456,172.493,26.305,154.806
C03577=1066.918,44.364,-68.440,172.492,26.302,154.805
C03578=1066.913,44.114,-68.423,172.490,26.299,154.805
C03579=1066.907,43.865,-68.407,172.489,26.297,154.805
C03580=1066.901,43.616,-68.390,172.487,26.294,154.804
C03581=1066.895,43.366,-68.374,172.486,26.291,154.804
C03582=1066.889,43.117,-68.358,172.485,26.289,154.804
C03583=1066.883,42.868,-68.342,172.484,26.286,154.803
C03584=1066.877,42.618,-68.325,172.483,26.283,154.803
C03585=1066.871,42.369,-68.309,172.481,26.280,154.803
C03586=1066.865,42.120,-68.293,172.480,26.278,154.802
C03587=1066.859,41.870,-68.277,172.478,26.275,154.802
C03588=1066.853,41.621,-68.260,172.477,26.272,154.801
C03589=1066.847,41.371,-68.245,172.475,26.270,154.801
C03590=1066.841,41.122,-68.228,172.474,26.267,154.801
C03591=1066.835,40.872,-68.212,172.473,26.264,154.800
C03592=1066.829,40.623,-68.197,172.471,26.262,154.800
C03593=1066.823,40.374,-68.180,172.470,26.259,154.800
C03594=1066.817,40.125,-68.164,172.468,26.256,154.799
C03595=1066.811,39.875,-68.148,172.467,26.254,154.799
C03596=1066.805,39.625,-68.132,172.465,26.251,154.799
C03597=1066.799,39.376,-68.116,172.464,26.248,154.798
C03598=1066.793,39.127,-68.100,172.463,26.245,154.798
C03599=1066.787,38.877,-68.083,172.461,26.243,154.798
C03600=1066.781,38.628,-68.067,172.460,26.240,154.797
C03601=1066.776,38.378,-68.052,172.458,26.237,154.797
C03602=1066.770,38.128,-68.035,172.457,26.235,154.797
C03603=1066.764,37.879,-68.019,172.456,26.232,154.796
C03604=1066.758,37.630,-68.003,172.454,26.229,154.796
C03605=1066.752,37.380,-67.988,172.453,26.227,154.795
C03606=1066.746,37.131,-67.972,172.451,26.224,154.795
C03607=1066.740,36.881,-67.955,172.450,26.222,154.795
C03608=1066.734,36.632,-67.939,172.448,26.219,154.794
C03609=1066.728,36.382,-67.924,172.447,26.216,154.794
C03610=1066.721,36.133,-67.908,172.446,26.214,154.794
C03611=1066.715,35.884,-67.892,172.445,26.211,154.793
C03612=1066.710,35.634,-67.875,172.443,26.209,154.793
C03613=1066.704,35.384,-67.860,172.442,26.206,154.793
C03614=1066.698,35.136,-67.845,172.441,26.203,154.792
C03615=1066.692,34.887,-67.828,172.439,26.201,154.792
C03616=1066.686,34.637,-67.813,172.438,26.198,154.792
C03617=1066.680,34.387,-67.797,172.436,26.195,154.791
C03618=1066.674,34.138,-67.781,172.435,26.193,154.791
C03619=1066.668,33.888,-67.765,172.434,26.190,154.790
C03620=1066.662,33.639,-67.749,172.432,26.188,154.790
C03621=1066.656,33.389,-67.734,172.431,26.185,154.790
C03622=1066.650,33.140,-67.718,172.429,26.182,154.789
C03623=1066.644,32.891,-67.702,172.428,26.180,154.789
C03624=1066.638,32.641,-67.686,172.426,26.177,154.789
C03625=1066.632,32.392,-67.671,172.425,26.174,154.788
C03626=1066.626,32.142,-67.655,172.423,26.172,154.788
C03627=1066.620,31.893,-67.639,172.422,26.169,154.788
